LIN {X 0,Y 368.953,Z 167.528,A -85,B 0,C 180,E1 -12752.796,E2 -12752.796} C_VEL
LIN {X 0,Y 368.922,Z 167.518,A -85,B 0,C 180,E1 -12756.117,E2 -12756.117} C_VEL
LIN {X 0,Y 368.919,Z 167.528,A -85,B 0,C 180,E1 -12759.946,E2 -12759.946} C_VEL
LIN {X 0,Y 368.957,Z 167.521,A -85,B 0,C 180,E1 -12763.398,E2 -12763.398} C_VEL
LIN {X 0,Y 369.049,Z 167.51,A -85,B 0,C 180,E1 -12766.79,E2 -12766.79} C_VEL
LIN {X 0,Y 369.059,Z 167.505,A -85,B 0,C 180,E1 -12770.132,E2 -12770.132} C_VEL
LIN {X 0,Y 369.151,Z 167.503,A -85,B 0,C 180,E1 -12772.342,E2 -12772.342} C_VEL
LIN {X 0,Y 369.129,Z 167.493,A -85,B 0,C 180,E1 -12774.537,E2 -12774.537} C_VEL
LIN {X 0,Y 369.304,Z 167.479,A -85,B 0,C 180,E1 -12777.819,E2 -12777.819} C_VEL
LIN {X 0,Y 369.446,Z 167.464,A -85,B 0,C 180,E1 -12780,E2 -12780} C_VEL
LIN {X 0,Y 369.303,Z 167.47,A -85,B 0,C 180,E1 -12782.181,E2 -12782.181} C_VEL
LIN {X 0,Y 369.185,Z 167.495,A -85,B 0,C 180,E1 -12786.687,E2 -12786.687} C_VEL
LIN {X 0,Y 369.126,Z 167.489,A -85,B 0,C 180,E1 -12788.761,E2 -12788.761} C_VEL
LIN {X 0,Y 368.994,Z 167.52,A -85,B 0,C 180,E1 -12792.094,E2 -12792.094} C_VEL
LIN {X 0,Y 368.987,Z 167.509,A -85,B 0,C 180,E1 -12795.465,E2 -12795.465} C_VEL
LIN {X 0,Y 368.956,Z 167.525,A -85,B 0,C 180,E1 -12798.894,E2 -12798.894} C_VEL
LIN {X 0,Y 368.922,Z 167.521,A -85,B 0,C 180,E1 -12802.396,E2 -12802.396} C_VEL
LIN {X 0,Y 368.991,Z 167.523,A -85,B 0,C 180,E1 -12805.981,E2 -12805.981} C_VEL
LIN {X 0,Y 368.95,Z 167.523,A -85,B 0,C 180,E1 -12808.812,E2 -12808.812} C_VEL
LIN {X 0,Y 368.89,Z 167.526,A -85,B 0,C 180,E1 -12812.239,E2 -12812.239} C_VEL
LIN {X 0,Y 368.921,Z 167.494,A -85,B 0,C 180,E1 -12815.002,E2 -12815.002} C_VEL
LIN {X 0,Y 368.901,Z 167.532,A -85,B 0,C 180,E1 -12818.641,E2 -12818.641} C_VEL
LIN {X 0,Y 368.875,Z 167.52,A -85,B 0,C 180,E1 -12822.01,E2 -12822.01} C_VEL
LIN {X 0,Y 368.874,Z 167.527,A -85,B 0,C 180,E1 -12825.177,E2 -12825.177} C_VEL
LIN {X 0,Y 368.878,Z 167.529,A -85,B 0,C 180,E1 -12828.179,E2 -12828.179} C_VEL
LIN {X 0,Y 368.902,Z 167.522,A -85,B 0,C 180,E1 -12831.361,E2 -12831.361} C_VEL
LIN {X 0,Y 368.933,Z 167.516,A -85,B 0,C 180,E1 -12835.148,E2 -12835.148} C_VEL
LIN {X 0,Y 368.927,Z 167.52,A -85,B 0,C 180,E1 -12839.048,E2 -12839.048} C_VEL
LIN {X 0,Y 368.975,Z 167.527,A -85,B 0,C 180,E1 -12842.799,E2 -12842.799} C_VEL
LIN {X 0,Y 369.055,Z 167.91,A -85,B 0,C 180,E1 -12843.213,E2 -12843.213} C_VEL
LIN {X 0,Y 371.306,Z 179.09,A -85,B 0,C 180,E1 -12846.304,E2 -12846.304} C_VEL
LIN {X 0,Y 372.031,Z 183.742,A -85,B 0,C 180,E1 -12847.54,E2 -12847.54} C_VEL
LIN {X 0,Y 371.856,Z 187.412,A -85,B 0,C 180,E1 -12848.395,E2 -12848.395} C_VEL
LIN {X 0,Y 374.592,Z 201.248,A -85,B 0,C 180,E1 -12848.88,E2 -12848.88} C_VEL
LIN {X 0,Y 377.012,Z 215.027,A -85,B 0,C 180,E1 -12849.298,E2 -12849.298} C_VEL
LIN {X 0,Y 375.8,Z 295.344,A -85,B 0,C 180,E1 -12850.862,E2 -12850.862} C_VEL
LIN {X 0,Y 375.266,Z 308.388,A -85,B 0,C 180,E1 -12851.33,E2 -12851.33} C_VEL
LIN {X 0,Y 374.412,Z 321.526,A -85,B 0,C 180,E1 -12852.029,E2 -12852.029} C_VEL
LIN {X 0,Y 373.468,Z 333.374,A -85,B 0,C 180,E1 -12852.901,E2 -12852.901} C_VEL
LIN {X 0,Y 372.421,Z 345.135,A -85,B 0,C 180,E1 -12854.022,E2 -12854.022} C_VEL
LIN {X 0,Y 371.58,Z 354.998,A -85,B 0,C 180,E1 -12855.207,E2 -12855.207} C_VEL
LIN {X 0,Y 370.573,Z 364.199,A -85,B 0,C 180,E1 -12856.567,E2 -12856.567} C_VEL
LIN {X 0,Y 369.519,Z 373.137,A -85,B 0,C 180,E1 -12858.203,E2 -12858.203} C_VEL
LIN {X 0,Y 368.777,Z 380.334,A -85,B 0,C 180,E1 -12859.847,E2 -12859.847} C_VEL
LIN {X 0,Y 368.263,Z 385.189,A -85,B 0,C 180,E1 -12861.219,E2 -12861.219} C_VEL
LIN {X 0,Y 367.893,Z 389.907,A -85,B 0,C 180,E1 -12862.868,E2 -12862.868} C_VEL
LIN {X 0,Y 367.658,Z 393.52,A -85,B 0,C 180,E1 -12864.516,E2 -12864.516} C_VEL
LIN {X 0,Y 367.551,Z 395.387,A -85,B 0,C 180,E1 -12865.614,E2 -12865.614} C_VEL
LIN {X 0,Y 367.409,Z 396.793,A -85,B 0,C 180,E1 -12866.711,E2 -12866.711} C_VEL
LIN {X 0,Y 367.36,Z 398.408,A -85,B 0,C 180,E1 -12868.904,E2 -12868.904} C_VEL
LIN {X 0,Y 367.375,Z 398.642,A -85,B 0,C 180,E1 -12870,E2 -12870} C_VEL
LIN {X 0,Y 367.36,Z 398.452,A -85,B 0,C 180,E1 -12871.097,E2 -12871.097} C_VEL
LIN {X 0,Y 367.408,Z 396.893,A -85,B 0,C 180,E1 -12873.29,E2 -12873.29} C_VEL
LIN {X 0,Y 367.547,Z 395.53,A -85,B 0,C 180,E1 -12874.387,E2 -12874.387} C_VEL
LIN {X 0,Y 367.757,Z 391.844,A -85,B 0,C 180,E1 -12876.411,E2 -12876.411} C_VEL
LIN {X 0,Y 368.118,Z 387.186,A -85,B 0,C 180,E1 -12878.233,E2 -12878.233} C_VEL
LIN {X 0,Y 368.737,Z 380.727,A -85,B 0,C 180,E1 -12880.155,E2 -12880.155} C_VEL
LIN {X 0,Y 369.473,Z 373.632,A -85,B 0,C 180,E1 -12881.799,E2 -12881.799} C_VEL
LIN {X 0,Y 370.503,Z 364.792,A -85,B 0,C 180,E1 -12883.437,E2 -12883.437} C_VEL
LIN {X 0,Y 371.506,Z 356.065,A -85,B 0,C 180,E1 -12884.747,E2 -12884.747} C_VEL
LIN {X 0,Y 372.173,Z 347.371,A -85,B 0,C 180,E1 -12885.835,E2 -12885.835} C_VEL
LIN {X 0,Y 373.258,Z 336.1,A -85,B 0,C 180,E1 -12886.969,E2 -12886.969} C_VEL
LIN {X 0,Y 373.899,Z 328.987,A -85,B 0,C 180,E1 -12887.548,E2 -12887.548} C_VEL
LIN {X 0,Y 373.639,Z 323.72,A -85,B 0,C 180,E1 -12887.96,E2 -12887.96} C_VEL
LIN {X 0,Y 371.467,Z 315.053,A -85,B 0,C 180,E1 -12888.627,E2 -12888.627} C_VEL
LIN {X 0,Y 369.299,Z 306.135,A -85,B 0,C 180,E1 -12889.198,E2 -12889.198} C_VEL
LIN {X 0,Y 368.949,Z 300.482,A -85,B 0,C 180,E1 -12889.447,E2 -12889.447} C_VEL
LIN {X 0,Y 369.32,Z 287.934,A -85,B 0,C 180,E1 -12889.778,E2 -12889.778} C_VEL
LIN {X 0,Y 370.382,Z 215.345,A -85,B 0,C 180,E1 -12891.19,E2 -12891.19} C_VEL
LIN {X 0,Y 365.229,Z 188.64,A -85,B 0,C 180,E1 -12892.066,E2 -12892.066} C_VEL
LIN {X 0,Y 365.048,Z 187.088,A -85,B 0,C 180,E1 -12892.199,E2 -12892.199} C_VEL
LIN {X 0,Y 364.993,Z 184.101,A -85,B 0,C 180,E1 -12892.949,E2 -12892.949} C_VEL
LIN {X 0,Y 362.795,Z 172.573,A -85,B 0,C 180,E1 -12896.149,E2 -12896.149} C_VEL
LIN {X 0,Y 361.954,Z 168.46,A -85,B 0,C 180,E1 -12897.396,E2 -12897.396} C_VEL
LIN {X 0,Y 361.847,Z 168.401,A -85,B 0,C 180,E1 -12901.285,E2 -12901.285} C_VEL
LIN {X 0,Y 361.855,Z 168.4,A -85,B 0,C 180,E1 -12904.28,E2 -12904.28} C_VEL
LIN {X 0,Y 361.863,Z 168.409,A -85,B 0,C 180,E1 -12907.222,E2 -12907.222} C_VEL
LIN {X 0,Y 361.834,Z 168.395,A -85,B 0,C 180,E1 -12910.755,E2 -12910.755} C_VEL
LIN {X 0,Y 361.815,Z 168.411,A -85,B 0,C 180,E1 -12914.368,E2 -12914.368} C_VEL
LIN {X 0,Y 361.834,Z 168.391,A -85,B 0,C 180,E1 -12917.568,E2 -12917.568} C_VEL
LIN {X 0,Y 361.868,Z 168.407,A -85,B 0,C 180,E1 -12920.973,E2 -12920.973} C_VEL
LIN {X 0,Y 361.872,Z 168.37,A -85,B 0,C 180,E1 -12924.655,E2 -12924.655} C_VEL
LIN {X 0,Y 361.835,Z 168.412,A -85,B 0,C 180,E1 -12928.37,E2 -12928.37} C_VEL
LIN {X 0,Y 361.897,Z 168.401,A -85,B 0,C 180,E1 -12930.955,E2 -12930.955} C_VEL
LIN {X 0,Y 361.95,Z 168.391,A -85,B 0,C 180,E1 -12933.475,E2 -12933.475} C_VEL
LIN {X 0,Y 361.875,Z 168.402,A -85,B 0,C 180,E1 -12937.144,E2 -12937.144} C_VEL
LIN {X 0,Y 361.905,Z 168.402,A -85,B 0,C 180,E1 -12940.723,E2 -12940.723} C_VEL
LIN {X 0,Y 361.928,Z 168.396,A -85,B 0,C 180,E1 -12943.066,E2 -12943.066} C_VEL
LIN {X 0,Y 361.994,Z 168.389,A -85,B 0,C 180,E1 -12946.528,E2 -12946.528} C_VEL
LIN {X 0,Y 362.026,Z 168.376,A -85,B 0,C 180,E1 -12949.938,E2 -12949.938} C_VEL
LIN {X 0,Y 362.145,Z 168.369,A -85,B 0,C 180,E1 -12952.192,E2 -12952.192} C_VEL
LIN {X 0,Y 362.109,Z 168.376,A -85,B 0,C 180,E1 -12954.431,E2 -12954.431} C_VEL
LIN {X 0,Y 362.273,Z 168.345,A -85,B 0,C 180,E1 -12957.776,E2 -12957.776} C_VEL
LIN {X 0,Y 362.42,Z 168.339,A -85,B 0,C 180,E1 -12960,E2 -12960} C_VEL
LIN {X 0,Y 362.274,Z 168.354,A -85,B 0,C 180,E1 -12962.224,E2 -12962.224} C_VEL
LIN {X 0,Y 362.142,Z 168.369,A -85,B 0,C 180,E1 -12966.687,E2 -12966.687} C_VEL
LIN {X 0,Y 361.994,Z 168.384,A -85,B 0,C 180,E1 -12970.063,E2 -12970.063} C_VEL
LIN {X 0,Y 361.993,Z 168.392,A -85,B 0,C 180,E1 -12973.899,E2 -12973.899} C_VEL
LIN {X 0,Y 361.923,Z 168.395,A -85,B 0,C 180,E1 -12976.934,E2 -12976.934} C_VEL
LIN {X 0,Y 361.878,Z 168.405,A -85,B 0,C 180,E1 -12980.461,E2 -12980.461} C_VEL
LIN {X 0,Y 361.889,Z 168.395,A -85,B 0,C 180,E1 -12984.113,E2 -12984.113} C_VEL
LIN {X 0,Y 361.937,Z 168.4,A -85,B 0,C 180,E1 -12986.722,E2 -12986.722} C_VEL
LIN {X 0,Y 361.869,Z 168.402,A -85,B 0,C 180,E1 -12990.328,E2 -12990.328} C_VEL
LIN {X 0,Y 361.851,Z 168.402,A -85,B 0,C 180,E1 -12994.281,E2 -12994.281} C_VEL
LIN {X 0,Y 361.859,Z 168.38,A -85,B 0,C 180,E1 -12997.223,E2 -12997.223} C_VEL
LIN {X 0,Y 361.832,Z 168.415,A -85,B 0,C 180,E1 -13000.756,E2 -13000.756} C_VEL
LIN {X 0,Y 361.814,Z 168.412,A -85,B 0,C 180,E1 -13004.369,E2 -13004.369} C_VEL
LIN {X 0,Y 361.829,Z 168.412,A -85,B 0,C 180,E1 -13007.57,E2 -13007.57} C_VEL
LIN {X 0,Y 361.826,Z 168.396,A -85,B 0,C 180,E1 -13010.982,E2 -13010.982} C_VEL
LIN {X 0,Y 361.874,Z 168.408,A -85,B 0,C 180,E1 -13014.656,E2 -13014.656} C_VEL
LIN {X 0,Y 361.838,Z 168.412,A -85,B 0,C 180,E1 -13018.371,E2 -13018.371} C_VEL
LIN {X 0,Y 361.881,Z 168.545,A -85,B 0,C 180,E1 -13021.271,E2 -13021.271} C_VEL
LIN {X 0,Y 364.14,Z 179.165,A -85,B 0,C 180,E1 -13024.262,E2 -13024.262} C_VEL
LIN {X 0,Y 365.433,Z 186.328,A -85,B 0,C 180,E1 -13026.18,E2 -13026.18} C_VEL
LIN {X 0,Y 364.841,Z 193.578,A -85,B 0,C 180,E1 -13027.899,E2 -13027.899} C_VEL
LIN {X 0,Y 368.892,Z 215.373,A -85,B 0,C 180,E1 -13028.637,E2 -13028.637} C_VEL
LIN {X 0,Y 370.384,Z 225.055,A -85,B 0,C 180,E1 -13028.924,E2 -13028.924} C_VEL
LIN {X 0,Y 369.098,Z 301.362,A -85,B 0,C 180,E1 -13030.427,E2 -13030.427} C_VEL
LIN {X 0,Y 368.43,Z 314.558,A -85,B 0,C 180,E1 -13030.897,E2 -13030.897} C_VEL
LIN {X 0,Y 367.598,Z 326.674,A -85,B 0,C 180,E1 -13031.539,E2 -13031.539} C_VEL
LIN {X 0,Y 366.61,Z 338.9,A -85,B 0,C 180,E1 -13032.426,E2 -13032.426} C_VEL
LIN {X 0,Y 365.481,Z 350.464,A -85,B 0,C 180,E1 -13033.523,E2 -13033.523} C_VEL
LIN {X 0,Y 364.402,Z 361.281,A -85,B 0,C 180,E1 -13034.819,E2 -13034.819} C_VEL
LIN {X 0,Y 363.383,Z 371.057,A -85,B 0,C 180,E1 -13036.295,E2 -13036.295} C_VEL
LIN {X 0,Y 362.293,Z 379.964,A -85,B 0,C 180,E1 -13037.963,E2 -13037.963} C_VEL
LIN {X 0,Y 361.542,Z 387.13,A -85,B 0,C 180,E1 -13039.641,E2 -13039.641} C_VEL
LIN {X 0,Y 360.902,Z 393.654,A -85,B 0,C 180,E1 -13041.602,E2 -13041.602} C_VEL
LIN {X 0,Y 360.576,Z 397.97,A -85,B 0,C 180,E1 -13043.284,E2 -13043.284} C_VEL
LIN {X 0,Y 360.446,Z 400.254,A -85,B 0,C 180,E1 -13044.405,E2 -13044.405} C_VEL
LIN {X 0,Y 360.388,Z 402.105,A -85,B 0,C 180,E1 -13045.526,E2 -13045.526} C_VEL
LIN {X 0,Y 360.286,Z 403.492,A -85,B 0,C 180,E1 -13046.645,E2 -13046.645} C_VEL
LIN {X 0,Y 360.249,Z 405.086,A -85,B 0,C 180,E1 -13048.882,E2 -13048.882} C_VEL
LIN {X 0,Y 360.274,Z 405.299,A -85,B 0,C 180,E1 -13050,E2 -13050} C_VEL
LIN {X 0,Y 360.249,Z 405.081,A -85,B 0,C 180,E1 -13051.117,E2 -13051.117} C_VEL
LIN {X 0,Y 360.286,Z 403.483,A -85,B 0,C 180,E1 -13053.354,E2 -13053.354} C_VEL
LIN {X 0,Y 360.388,Z 402.092,A -85,B 0,C 180,E1 -13054.473,E2 -13054.473} C_VEL
LIN {X 0,Y 360.51,Z 399.158,A -85,B 0,C 180,E1 -13056.159,E2 -13056.159} C_VEL
LIN {X 0,Y 360.775,Z 395.206,A -85,B 0,C 180,E1 -13057.837,E2 -13057.837} C_VEL
LIN {X 0,Y 361.306,Z 389.114,A -85,B 0,C 180,E1 -13059.799,E2 -13059.799} C_VEL
LIN {X 0,Y 362.024,Z 382.458,A -85,B 0,C 180,E1 -13061.477,E2 -13061.477} C_VEL
LIN {X 0,Y 362.976,Z 374.197,A -85,B 0,C 180,E1 -13063.149,E2 -13063.149} C_VEL
LIN {X 0,Y 363.939,Z 365.725,A -85,B 0,C 180,E1 -13064.538,E2 -13064.538} C_VEL
LIN {X 0,Y 364.962,Z 355.253,A -85,B 0,C 180,E1 -13065.926,E2 -13065.926} C_VEL
LIN {X 0,Y 366.116,Z 343.462,A -85,B 0,C 180,E1 -13067.165,E2 -13067.165} C_VEL
LIN {X 0,Y 367.216,Z 331.594,A -85,B 0,C 180,E1 -13068.119,E2 -13068.119} C_VEL
LIN {X 0,Y 368.176,Z 319.239,A -85,B 0,C 180,E1 -13068.863,E2 -13068.863} C_VEL
LIN {X 0,Y 368.825,Z 306.535,A -85,B 0,C 180,E1 -13069.406,E2 -13069.406} C_VEL
LIN {X 0,Y 369.28,Z 293.176,A -85,B 0,C 180,E1 -13069.743,E2 -13069.743} C_VEL
LIN {X 0,Y 370.205,Z 223.387,A -85,B 0,C 180,E1 -13071.106,E2 -13071.106} C_VEL
LIN {X 0,Y 365.253,Z 196.039,A -85,B 0,C 180,E1 -13071.971,E2 -13071.971} C_VEL
LIN {X 0,Y 364.814,Z 193.463,A -85,B 0,C 180,E1 -13072.102,E2 -13072.102} C_VEL
LIN {X 0,Y 365.418,Z 186.266,A -85,B 0,C 180,E1 -13073.82,E2 -13073.82} C_VEL
LIN {X 0,Y 363.121,Z 174.181,A -85,B 0,C 180,E1 -13077.088,E2 -13077.088} C_VEL
LIN {X 0,Y 361.886,Z 168.471,A -85,B 0,C 180,E1 -13078.756,E2 -13078.756} C_VEL
LIN {X 0,Y 361.835,Z 168.413,A -85,B 0,C 180,E1 -13081.628,E2 -13081.628} C_VEL
LIN {X 0,Y 361.87,Z 168.409,A -85,B 0,C 180,E1 -13085.344,E2 -13085.344} C_VEL
LIN {X 0,Y 361.824,Z 168.397,A -85,B 0,C 180,E1 -13089.017,E2 -13089.017} C_VEL
LIN {X 0,Y 361.83,Z 168.409,A -85,B 0,C 180,E1 -13092.828,E2 -13092.828} C_VEL
LIN {X 0,Y 361.812,Z 168.411,A -85,B 0,C 180,E1 -13095.946,E2 -13095.946} C_VEL
LIN {X 0,Y 361.828,Z 168.415,A -85,B 0,C 180,E1 -13099.244,E2 -13099.244} C_VEL
LIN {X 0,Y 361.855,Z 168.38,A -85,B 0,C 180,E1 -13102.776,E2 -13102.776} C_VEL
LIN {X 0,Y 361.846,Z 168.404,A -85,B 0,C 180,E1 -13105.719,E2 -13105.719} C_VEL
LIN {X 0,Y 361.864,Z 168.402,A -85,B 0,C 180,E1 -13109.671,E2 -13109.671} C_VEL
LIN {X 0,Y 361.944,Z 168.398,A -85,B 0,C 180,E1 -13113.474,E2 -13113.474} C_VEL
LIN {X 0,Y 361.869,Z 168.405,A -85,B 0,C 180,E1 -13117.143,E2 -13117.143} C_VEL
LIN {X 0,Y 361.891,Z 168.4,A -85,B 0,C 180,E1 -13120.722,E2 -13120.722} C_VEL
LIN {X 0,Y 361.933,Z 168.397,A -85,B 0,C 180,E1 -13124.226,E2 -13124.226} C_VEL
LIN {X 0,Y 361.99,Z 168.392,A -85,B 0,C 180,E1 -13126.527,E2 -13126.527} C_VEL
LIN {X 0,Y 362.023,Z 168.381,A -85,B 0,C 180,E1 -13129.938,E2 -13129.938} C_VEL
LIN {X 0,Y 362.149,Z 168.368,A -85,B 0,C 180,E1 -13133.313,E2 -13133.313} C_VEL
LIN {X 0,Y 362.268,Z 168.355,A -85,B 0,C 180,E1 -13137.776,E2 -13137.776} C_VEL
LIN {X 0,Y 362.416,Z 168.34,A -85,B 0,C 180,E1 -13140,E2 -13140} C_VEL
LIN {X 0,Y 362.268,Z 168.346,A -85,B 0,C 180,E1 -13142.224,E2 -13142.224} C_VEL
LIN {X 0,Y 362.158,Z 168.37,A -85,B 0,C 180,E1 -13146.686,E2 -13146.686} C_VEL
LIN {X 0,Y 362.063,Z 168.368,A -85,B 0,C 180,E1 -13148.934,E2 -13148.934} C_VEL
LIN {X 0,Y 361.949,Z 168.4,A -85,B 0,C 180,E1 -13152.333,E2 -13152.333} C_VEL
LIN {X 0,Y 361.951,Z 168.388,A -85,B 0,C 180,E1 -13154.621,E2 -13154.621} C_VEL
LIN {X 0,Y 361.947,Z 168.397,A -85,B 0,C 180,E1 -13158.1,E2 -13158.1} C_VEL
LIN {X 0,Y 361.882,Z 168.398,A -85,B 0,C 180,E1 -13161.654,E2 -13161.654} C_VEL
LIN {X 0,Y 361.919,Z 168.401,A -85,B 0,C 180,E1 -13165.291,E2 -13165.291} C_VEL
LIN {X 0,Y 361.905,Z 168.395,A -85,B 0,C 180,E1 -13167.779,E2 -13167.779} C_VEL
LIN {X 0,Y 361.839,Z 168.41,A -85,B 0,C 180,E1 -13171.286,E2 -13171.286} C_VEL
LIN {X 0,Y 361.846,Z 168.379,A -85,B 0,C 180,E1 -13174.281,E2 -13174.281} C_VEL
LIN {X 0,Y 361.856,Z 168.396,A -85,B 0,C 180,E1 -13177.224,E2 -13177.224} C_VEL
LIN {X 0,Y 361.829,Z 168.409,A -85,B 0,C 180,E1 -13180.756,E2 -13180.756} C_VEL
LIN {X 0,Y 361.81,Z 168.396,A -85,B 0,C 180,E1 -13184.37,E2 -13184.37} C_VEL
LIN {X 0,Y 361.831,Z 168.415,A -85,B 0,C 180,E1 -13187.569,E2 -13187.569} C_VEL
LIN {X 0,Y 361.864,Z 168.394,A -85,B 0,C 180,E1 -13190.975,E2 -13190.975} C_VEL
LIN {X 0,Y 361.871,Z 168.397,A -85,B 0,C 180,E1 -13194.656,E2 -13194.656} C_VEL
LIN {X 0,Y 361.835,Z 168.405,A -85,B 0,C 180,E1 -13198.372,E2 -13198.372} C_VEL
LIN {X 0,Y 361.913,Z 168.401,A -85,B 0,C 180,E1 -13202.223,E2 -13202.223} C_VEL
LIN {X 0,Y 361.98,Z 168.589,A -85,B 0,C 180,E1 -13202.791,E2 -13202.791} C_VEL
LIN {X 0,Y 364.016,Z 178.714,A -85,B 0,C 180,E1 -13205.683,E2 -13205.683} C_VEL
LIN {X 0,Y 365.086,Z 185.481,A -85,B 0,C 180,E1 -13207.521,E2 -13207.521} C_VEL
LIN {X 0,Y 365.036,Z 187.672,A -85,B 0,C 180,E1 -13207.989,E2 -13207.989} C_VEL
LIN {X 0,Y 370.137,Z 213.867,A -85,B 0,C 180,E1 -13208.87,E2 -13208.87} C_VEL
LIN {X 0,Y 370.357,Z 219.609,A -85,B 0,C 180,E1 -13209,E2 -13209} C_VEL
LIN {X 0,Y 369.118,Z 295.425,A -85,B 0,C 180,E1 -13210.502,E2 -13210.502} C_VEL
LIN {X 0,Y 368.552,Z 308.464,A -85,B 0,C 180,E1 -13210.977,E2 -13210.977} C_VEL
LIN {X 0,Y 367.782,Z 320.497,A -85,B 0,C 180,E1 -13211.622,E2 -13211.622} C_VEL
LIN {X 0,Y 366.817,Z 331.857,A -85,B 0,C 180,E1 -13212.438,E2 -13212.438} C_VEL
LIN {X 0,Y 365.721,Z 343.786,A -85,B 0,C 180,E1 -13213.564,E2 -13213.564} C_VEL
LIN {X 0,Y 364.784,Z 354.024,A -85,B 0,C 180,E1 -13214.785,E2 -13214.785} C_VEL
LIN {X 0,Y 363.837,Z 362.569,A -85,B 0,C 180,E1 -13216.028,E2 -13216.028} C_VEL
LIN {X 0,Y 362.915,Z 370.46,A -85,B 0,C 180,E1 -13217.417,E2 -13217.417} C_VEL
LIN {X 0,Y 362.007,Z 378.174,A -85,B 0,C 180,E1 -13219.09,E2 -13219.09} C_VEL
LIN {X 0,Y 361.242,Z 385.256,A -85,B 0,C 180,E1 -13221.047,E2 -13221.047} C_VEL
LIN {X 0,Y 360.842,Z 389.973,A -85,B 0,C 180,E1 -13222.728,E2 -13222.728} C_VEL
LIN {X 0,Y 360.573,Z 393.586,A -85,B 0,C 180,E1 -13224.408,E2 -13224.408} C_VEL
LIN {X 0,Y 360.486,Z 395.452,A -85,B 0,C 180,E1 -13225.528,E2 -13225.528} C_VEL
LIN {X 0,Y 360.332,Z 396.859,A -85,B 0,C 180,E1 -13226.646,E2 -13226.646} C_VEL
LIN {X 0,Y 360.26,Z 398.474,A -85,B 0,C 180,E1 -13228.883,E2 -13228.883} C_VEL
LIN {X 0,Y 360.275,Z 398.707,A -85,B 0,C 180,E1 -13230,E2 -13230} C_VEL
LIN {X 0,Y 360.26,Z 398.517,A -85,B 0,C 180,E1 -13231.118,E2 -13231.118} C_VEL
LIN {X 0,Y 360.33,Z 396.958,A -85,B 0,C 180,E1 -13233.355,E2 -13233.355} C_VEL
LIN {X 0,Y 360.459,Z 395.595,A -85,B 0,C 180,E1 -13234.473,E2 -13234.473} C_VEL
LIN {X 0,Y 360.684,Z 392.187,A -85,B 0,C 180,E1 -13236.41,E2 -13236.41} C_VEL
LIN {X 0,Y 361.078,Z 387.25,A -85,B 0,C 180,E1 -13238.394,E2 -13238.394} C_VEL
LIN {X 0,Y 361.739,Z 380.79,A -85,B 0,C 180,E1 -13240.353,E2 -13240.353} C_VEL
LIN {X 0,Y 362.487,Z 373.695,A -85,B 0,C 180,E1 -13242.03,E2 -13242.03} C_VEL
LIN {X 0,Y 363.584,Z 364.854,A -85,B 0,C 180,E1 -13243.697,E2 -13243.697} C_VEL
LIN {X 0,Y 364.718,Z 355.058,A -85,B 0,C 180,E1 -13245.183,E2 -13245.183} C_VEL
LIN {X 0,Y 365.509,Z 345.747,A -85,B 0,C 180,E1 -13246.332,E2 -13246.332} C_VEL
LIN {X 0,Y 366.609,Z 334.579,A -85,B 0,C 180,E1 -13247.43,E2 -13247.43} C_VEL
LIN {X 0,Y 367.68,Z 322.048,A -85,B 0,C 180,E1 -13248.384,E2 -13248.384} C_VEL
LIN {X 0,Y 368.487,Z 309.138,A -85,B 0,C 180,E1 -13249.1,E2 -13249.1} C_VEL
LIN {X 0,Y 368.949,Z 300.482,A -85,B 0,C 180,E1 -13249.447,E2 -13249.447} C_VEL
LIN {X 0,Y 368.568,Z 294.756,A -85,B 0,C 180,E1 -13249.661,E2 -13249.661} C_VEL
LIN {X 0,Y 363.474,Z 276.11,A -85,B 0,C 180,E1 -13250.361,E2 -13250.361} C_VEL
LIN {X 0,Y 362.943,Z 270.294,A -85,B 0,C 180,E1 -13250.505,E2 -13250.505} C_VEL
LIN {X 0,Y 363.768,Z 216.155,A -85,B 0,C 180,E1 -13251.579,E2 -13251.579} C_VEL
LIN {X 0,Y 358.454,Z 188.842,A -85,B 0,C 180,E1 -13252.5,E2 -13252.5} C_VEL
LIN {X 0,Y 358.231,Z 187.146,A -85,B 0,C 180,E1 -13252.646,E2 -13252.646} C_VEL
LIN {X 0,Y 356.625,Z 177.642,A -85,B 0,C 180,E1 -13255.272,E2 -13255.272} C_VEL
LIN {X 0,Y 354.899,Z 169.377,A -85,B 0,C 180,E1 -13257.733,E2 -13257.733} C_VEL
LIN {X 0,Y 354.8,Z 169.28,A -85,B 0,C 180,E1 -13260.998,E2 -13260.998} C_VEL
LIN {X 0,Y 354.807,Z 169.285,A -85,B 0,C 180,E1 -13263.702,E2 -13263.702} C_VEL
LIN {X 0,Y 354.798,Z 169.287,A -85,B 0,C 180,E1 -13266.459,E2 -13266.459} C_VEL
LIN {X 0,Y 354.824,Z 169.267,A -85,B 0,C 180,E1 -13269.423,E2 -13269.423} C_VEL
LIN {X 0,Y 354.787,Z 169.29,A -85,B 0,C 180,E1 -13272.867,E2 -13272.867} C_VEL
LIN {X 0,Y 354.764,Z 169.27,A -85,B 0,C 180,E1 -13276.103,E2 -13276.103} C_VEL
LIN {X 0,Y 354.786,Z 169.286,A -85,B 0,C 180,E1 -13279.179,E2 -13279.179} C_VEL
LIN {X 0,Y 354.805,Z 169.278,A -85,B 0,C 180,E1 -13282.402,E2 -13282.402} C_VEL
LIN {X 0,Y 354.809,Z 169.248,A -85,B 0,C 180,E1 -13284.94,E2 -13284.94} C_VEL
LIN {X 0,Y 354.79,Z 169.29,A -85,B 0,C 180,E1 -13288.405,E2 -13288.405} C_VEL
LIN {X 0,Y 354.846,Z 169.278,A -85,B 0,C 180,E1 -13291.618,E2 -13291.618} C_VEL
LIN {X 0,Y 354.894,Z 169.279,A -85,B 0,C 180,E1 -13294.172,E2 -13294.172} C_VEL
LIN {X 0,Y 354.811,Z 169.277,A -85,B 0,C 180,E1 -13297.892,E2 -13297.892} C_VEL
LIN {X 0,Y 354.919,Z 169.273,A -85,B 0,C 180,E1 -13301.891,E2 -13301.891} C_VEL
LIN {X 0,Y 354.938,Z 169.269,A -85,B 0,C 180,E1 -13305.981,E2 -13305.981} C_VEL
LIN {X 0,Y 354.972,Z 169.256,A -85,B 0,C 180,E1 -13309.736,E2 -13309.736} C_VEL
LIN {X 0,Y 355.108,Z 169.243,A -85,B 0,C 180,E1 -13312.037,E2 -13312.037} C_VEL
LIN {X 0,Y 355.084,Z 169.251,A -85,B 0,C 180,E1 -13314.32,E2 -13314.32} C_VEL
LIN {X 0,Y 355.236,Z 169.221,A -85,B 0,C 180,E1 -13317.732,E2 -13317.732} C_VEL
LIN {X 0,Y 355.369,Z 169.218,A -85,B 0,C 180,E1 -13320,E2 -13320} C_VEL
LIN {X 0,Y 355.237,Z 169.231,A -85,B 0,C 180,E1 -13322.268,E2 -13322.268} C_VEL
LIN {X 0,Y 355.105,Z 169.246,A -85,B 0,C 180,E1 -13326.82,E2 -13326.82} C_VEL
LIN {X 0,Y 354.95,Z 169.261,A -85,B 0,C 180,E1 -13330.265,E2 -13330.265} C_VEL
LIN {X 0,Y 354.938,Z 169.271,A -85,B 0,C 180,E1 -13334.019,E2 -13334.019} C_VEL
LIN {X 0,Y 354.885,Z 169.266,A -85,B 0,C 180,E1 -13338.092,E2 -13338.092} C_VEL
LIN {X 0,Y 354.811,Z 169.284,A -85,B 0,C 180,E1 -13342.108,E2 -13342.108} C_VEL
LIN {X 0,Y 354.894,Z 169.277,A -85,B 0,C 180,E1 -13345.828,E2 -13345.828} C_VEL
LIN {X 0,Y 354.814,Z 169.28,A -85,B 0,C 180,E1 -13349.682,E2 -13349.682} C_VEL
LIN {X 0,Y 354.803,Z 169.281,A -85,B 0,C 180,E1 -13353.702,E2 -13353.702} C_VEL
LIN {X 0,Y 354.794,Z 169.256,A -85,B 0,C 180,E1 -13356.46,E2 -13356.46} C_VEL
LIN {X 0,Y 354.822,Z 169.283,A -85,B 0,C 180,E1 -13359.424,E2 -13359.424} C_VEL
LIN {X 0,Y 354.785,Z 169.284,A -85,B 0,C 180,E1 -13362.867,E2 -13362.867} C_VEL
LIN {X 0,Y 354.764,Z 169.292,A -85,B 0,C 180,E1 -13366.104,E2 -13366.104} C_VEL
LIN {X 0,Y 354.78,Z 169.291,A -85,B 0,C 180,E1 -13369.178,E2 -13369.178} C_VEL
LIN {X 0,Y 354.799,Z 169.274,A -85,B 0,C 180,E1 -13372.404,E2 -13372.404} C_VEL
LIN {X 0,Y 354.811,Z 169.283,A -85,B 0,C 180,E1 -13374.941,E2 -13374.941} C_VEL
LIN {X 0,Y 354.794,Z 169.289,A -85,B 0,C 180,E1 -13378.405,E2 -13378.405} C_VEL
LIN {X 0,Y 354.842,Z 169.383,A -85,B 0,C 180,E1 -13380.883,E2 -13380.883} C_VEL
LIN {X 0,Y 357.171,Z 180.29,A -85,B 0,C 180,E1 -13384.036,E2 -13384.036} C_VEL
LIN {X 0,Y 358.462,Z 187.453,A -85,B 0,C 180,E1 -13385.995,E2 -13385.995} C_VEL
LIN {X 0,Y 358.046,Z 193.292,A -85,B 0,C 180,E1 -13387.429,E2 -13387.429} C_VEL
LIN {X 0,Y 358.746,Z 197.435,A -85,B 0,C 180,E1 -13387.623,E2 -13387.623} C_VEL
LIN {X 0,Y 363.292,Z 222.248,A -85,B 0,C 180,E1 -13388.435,E2 -13388.435} C_VEL
LIN {X 0,Y 363.756,Z 226.414,A -85,B 0,C 180,E1 -13388.55,E2 -13388.55} C_VEL
LIN {X 0,Y 362.423,Z 301.31,A -85,B 0,C 180,E1 -13390.052,E2 -13390.052} C_VEL
LIN {X 0,Y 361.734,Z 314.502,A -85,B 0,C 180,E1 -13390.529,E2 -13390.529} C_VEL
LIN {X 0,Y 360.875,Z 326.615,A -85,B 0,C 180,E1 -13391.183,E2 -13391.183} C_VEL
LIN {X 0,Y 359.841,Z 338.839,A -85,B 0,C 180,E1 -13392.085,E2 -13392.085} C_VEL
LIN {X 0,Y 358.669,Z 350.403,A -85,B 0,C 180,E1 -13393.201,E2 -13393.201} C_VEL
LIN {X 0,Y 357.539,Z 361.219,A -85,B 0,C 180,E1 -13394.521,E2 -13394.521} C_VEL
LIN {X 0,Y 356.484,Z 370.994,A -85,B 0,C 180,E1 -13396.024,E2 -13396.024} C_VEL
LIN {X 0,Y 355.311,Z 379.9,A -85,B 0,C 180,E1 -13397.723,E2 -13397.723} C_VEL
LIN {X 0,Y 354.521,Z 387.066,A -85,B 0,C 180,E1 -13399.434,E2 -13399.434} C_VEL
LIN {X 0,Y 353.853,Z 393.59,A -85,B 0,C 180,E1 -13401.433,E2 -13401.433} C_VEL
LIN {X 0,Y 353.509,Z 397.905,A -85,B 0,C 180,E1 -13403.149,E2 -13403.149} C_VEL
LIN {X 0,Y 353.357,Z 400.19,A -85,B 0,C 180,E1 -13404.292,E2 -13404.292} C_VEL
LIN {X 0,Y 353.303,Z 402.041,A -85,B 0,C 180,E1 -13405.436,E2 -13405.436} C_VEL
LIN {X 0,Y 353.211,Z 403.428,A -85,B 0,C 180,E1 -13406.577,E2 -13406.577} C_VEL
LIN {X 0,Y 353.148,Z 405.021,A -85,B 0,C 180,E1 -13408.859,E2 -13408.859} C_VEL
LIN {X 0,Y 353.175,Z 405.234,A -85,B 0,C 180,E1 -13410,E2 -13410} C_VEL
LIN {X 0,Y 353.148,Z 405.016,A -85,B 0,C 180,E1 -13411.14,E2 -13411.14} C_VEL
LIN {X 0,Y 353.21,Z 403.418,A -85,B 0,C 180,E1 -13413.422,E2 -13413.422} C_VEL
LIN {X 0,Y 353.303,Z 402.026,A -85,B 0,C 180,E1 -13414.563,E2 -13414.563} C_VEL
LIN {X 0,Y 353.434,Z 399.342,A -85,B 0,C 180,E1 -13416.149,E2 -13416.149} C_VEL
LIN {X 0,Y 353.723,Z 395.14,A -85,B 0,C 180,E1 -13417.994,E2 -13417.994} C_VEL
LIN {X 0,Y 354.29,Z 389.048,A -85,B 0,C 180,E1 -13419.995,E2 -13419.995} C_VEL
LIN {X 0,Y 355.022,Z 382.391,A -85,B 0,C 180,E1 -13421.706,E2 -13421.706} C_VEL
LIN {X 0,Y 356.048,Z 374.13,A -85,B 0,C 180,E1 -13423.41,E2 -13423.41} C_VEL
LIN {X 0,Y 357.043,Z 365.658,A -85,B 0,C 180,E1 -13424.825,E2 -13424.825} C_VEL
LIN {X 0,Y 358.13,Z 355.185,A -85,B 0,C 180,E1 -13426.238,E2 -13426.238} C_VEL
LIN {X 0,Y 359.339,Z 343.393,A -85,B 0,C 180,E1 -13427.499,E2 -13427.499} C_VEL
LIN {X 0,Y 360.483,Z 331.523,A -85,B 0,C 180,E1 -13428.469,E2 -13428.469} C_VEL
LIN {X 0,Y 361.446,Z 319.166,A -85,B 0,C 180,E1 -13429.227,E2 -13429.227} C_VEL
LIN {X 0,Y 362.133,Z 306.459,A -85,B 0,C 180,E1 -13429.779,E2 -13429.779} C_VEL
LIN {X 0,Y 362.612,Z 293.091,A -85,B 0,C 180,E1 -13430.121,E2 -13430.121} C_VEL
LIN {X 0,Y 363.594,Z 224.394,A -85,B 0,C 180,E1 -13431.486,E2 -13431.486} C_VEL
LIN {X 0,Y 358.821,Z 197.843,A -85,B 0,C 180,E1 -13432.346,E2 -13432.346} C_VEL
LIN {X 0,Y 358.017,Z 193.627,A -85,B 0,C 180,E1 -13432.516,E2 -13432.516} C_VEL
LIN {X 0,Y 358.48,Z 188.58,A -85,B 0,C 180,E1 -13433.696,E2 -13433.696} C_VEL
LIN {X 0,Y 357.359,Z 181.416,A -85,B 0,C 180,E1 -13435.635,E2 -13435.635} C_VEL
LIN {X 0,Y 355.129,Z 170.735,A -85,B 0,C 180,E1 -13438.657,E2 -13438.657} C_VEL
LIN {X 0,Y 354.808,Z 169.313,A -85,B 0,C 180,E1 -13439.152,E2 -13439.152} C_VEL
LIN {X 0,Y 354.784,Z 169.294,A -85,B 0,C 180,E1 -13442.332,E2 -13442.332} C_VEL
LIN {X 0,Y 354.818,Z 169.289,A -85,B 0,C 180,E1 -13445.698,E2 -13445.698} C_VEL
LIN {X 0,Y 354.794,Z 169.276,A -85,B 0,C 180,E1 -13449.417,E2 -13449.417} C_VEL
LIN {X 0,Y 354.782,Z 169.287,A -85,B 0,C 180,E1 -13452.866,E2 -13452.866} C_VEL
LIN {X 0,Y 354.76,Z 169.289,A -85,B 0,C 180,E1 -13456.102,E2 -13456.102} C_VEL
LIN {X 0,Y 354.781,Z 169.293,A -85,B 0,C 180,E1 -13459.178,E2 -13459.178} C_VEL
LIN {X 0,Y 354.799,Z 169.261,A -85,B 0,C 180,E1 -13462.402,E2 -13462.402} C_VEL
LIN {X 0,Y 354.803,Z 169.266,A -85,B 0,C 180,E1 -13464.94,E2 -13464.94} C_VEL
LIN {X 0,Y 354.785,Z 169.291,A -85,B 0,C 180,E1 -13468.404,E2 -13468.404} C_VEL
LIN {X 0,Y 354.837,Z 169.281,A -85,B 0,C 180,E1 -13471.618,E2 -13471.618} C_VEL
LIN {X 0,Y 354.888,Z 169.277,A -85,B 0,C 180,E1 -13474.172,E2 -13474.172} C_VEL
LIN {X 0,Y 354.805,Z 169.285,A -85,B 0,C 180,E1 -13477.892,E2 -13477.892} C_VEL
LIN {X 0,Y 354.879,Z 169.266,A -85,B 0,C 180,E1 -13481.907,E2 -13481.907} C_VEL
LIN {X 0,Y 354.933,Z 169.271,A -85,B 0,C 180,E1 -13485.981,E2 -13485.981} C_VEL
LIN {X 0,Y 354.97,Z 169.259,A -85,B 0,C 180,E1 -13489.736,E2 -13489.736} C_VEL
LIN {X 0,Y 355.114,Z 169.245,A -85,B 0,C 180,E1 -13493.18,E2 -13493.18} C_VEL
LIN {X 0,Y 355.231,Z 169.232,A -85,B 0,C 180,E1 -13497.732,E2 -13497.732} C_VEL
LIN {X 0,Y 355.385,Z 169.215,A -85,B 0,C 180,E1 -13500,E2 -13500} C_VEL
LIN {X 0,Y 355.231,Z 169.222,A -85,B 0,C 180,E1 -13502.268,E2 -13502.268} C_VEL
LIN {X 0,Y 355.125,Z 169.245,A -85,B 0,C 180,E1 -13506.82,E2 -13506.82} C_VEL
LIN {X 0,Y 355.004,Z 169.246,A -85,B 0,C 180,E1 -13509.113,E2 -13509.113} C_VEL
LIN {X 0,Y 354.91,Z 169.276,A -85,B 0,C 180,E1 -13512.581,E2 -13512.581} C_VEL
LIN {X 0,Y 354.879,Z 169.266,A -85,B 0,C 180,E1 -13516.097,E2 -13516.097} C_VEL
LIN {X 0,Y 354.893,Z 169.28,A -85,B 0,C 180,E1 -13518.473,E2 -13518.473} C_VEL
LIN {X 0,Y 354.825,Z 169.276,A -85,B 0,C 180,E1 -13522.107,E2 -13522.107} C_VEL
LIN {X 0,Y 354.89,Z 169.279,A -85,B 0,C 180,E1 -13525.828,E2 -13525.828} C_VEL
LIN {X 0,Y 354.845,Z 169.281,A -85,B 0,C 180,E1 -13529.68,E2 -13529.68} C_VEL
LIN {X 0,Y 354.799,Z 169.264,A -85,B 0,C 180,E1 -13533.703,E2 -13533.703} C_VEL
LIN {X 0,Y 354.79,Z 169.262,A -85,B 0,C 180,E1 -13536.461,E2 -13536.461} C_VEL
LIN {X 0,Y 354.818,Z 169.286,A -85,B 0,C 180,E1 -13539.425,E2 -13539.425} C_VEL
LIN {X 0,Y 354.782,Z 169.267,A -85,B 0,C 180,E1 -13542.868,E2 -13542.868} C_VEL
LIN {X 0,Y 354.762,Z 169.293,A -85,B 0,C 180,E1 -13546.105,E2 -13546.105} C_VEL
LIN {X 0,Y 354.782,Z 169.276,A -85,B 0,C 180,E1 -13549.18,E2 -13549.18} C_VEL
LIN {X 0,Y 354.803,Z 169.29,A -85,B 0,C 180,E1 -13552.404,E2 -13552.404} C_VEL
LIN {X 0,Y 354.809,Z 169.275,A -85,B 0,C 180,E1 -13554.942,E2 -13554.942} C_VEL
LIN {X 0,Y 354.791,Z 169.282,A -85,B 0,C 180,E1 -13558.406,E2 -13558.406} C_VEL
LIN {X 0,Y 354.848,Z 169.278,A -85,B 0,C 180,E1 -13561.62,E2 -13561.62} C_VEL
LIN {X 0,Y 354.92,Z 169.503,A -85,B 0,C 180,E1 -13562.446,E2 -13562.446} C_VEL
LIN {X 0,Y 357.111,Z 180.301,A -85,B 0,C 180,E1 -13565.59,E2 -13565.59} C_VEL
LIN {X 0,Y 358.159,Z 187.07,A -85,B 0,C 180,E1 -13567.439,E2 -13567.439} C_VEL
LIN {X 0,Y 358.218,Z 187.932,A -85,B 0,C 180,E1 -13567.561,E2 -13567.561} C_VEL
LIN {X 0,Y 363.054,Z 212.192,A -85,B 0,C 180,E1 -13568.4,E2 -13568.4} C_VEL
LIN {X 0,Y 363.803,Z 217.381,A -85,B 0,C 180,E1 -13568.555,E2 -13568.555} C_VEL
LIN {X 0,Y 362.454,Z 295.506,A -85,B 0,C 180,E1 -13570.128,E2 -13570.128} C_VEL
LIN {X 0,Y 361.839,Z 308.539,A -85,B 0,C 180,E1 -13570.61,E2 -13570.61} C_VEL
LIN {X 0,Y 361.043,Z 320.57,A -85,B 0,C 180,E1 -13571.266,E2 -13571.266} C_VEL
LIN {X 0,Y 360.059,Z 331.928,A -85,B 0,C 180,E1 -13572.097,E2 -13572.097} C_VEL
LIN {X 0,Y 358.919,Z 343.855,A -85,B 0,C 180,E1 -13573.243,E2 -13573.243} C_VEL
LIN {X 0,Y 357.921,Z 353.931,A -85,B 0,C 180,E1 -13574.464,E2 -13574.464} C_VEL
LIN {X 0,Y 356.953,Z 362.637,A -85,B 0,C 180,E1 -13575.753,E2 -13575.753} C_VEL
LIN {X 0,Y 355.977,Z 370.527,A -85,B 0,C 180,E1 -13577.168,E2 -13577.168} C_VEL
LIN {X 0,Y 355.024,Z 378.241,A -85,B 0,C 180,E1 -13578.872,E2 -13578.872} C_VEL
LIN {X 0,Y 354.447,Z 383.507,A -85,B 0,C 180,E1 -13580.298,E2 -13580.298} C_VEL
LIN {X 0,Y 353.911,Z 388.617,A -85,B 0,C 180,E1 -13582.01,E2 -13582.01} C_VEL
LIN {X 0,Y 353.591,Z 392.373,A -85,B 0,C 180,E1 -13583.621,E2 -13583.621} C_VEL
LIN {X 0,Y 353.4,Z 395.518,A -85,B 0,C 180,E1 -13585.438,E2 -13585.438} C_VEL
LIN {X 0,Y 353.257,Z 396.924,A -85,B 0,C 180,E1 -13586.579,E2 -13586.579} C_VEL
LIN {X 0,Y 353.16,Z 398.539,A -85,B 0,C 180,E1 -13588.86,E2 -13588.86} C_VEL
LIN {X 0,Y 353.176,Z 398.772,A -85,B 0,C 180,E1 -13590,E2 -13590} C_VEL
LIN {X 0,Y 353.16,Z 398.582,A -85,B 0,C 180,E1 -13591.141,E2 -13591.141} C_VEL
LIN {X 0,Y 353.254,Z 397.022,A -85,B 0,C 180,E1 -13593.422,E2 -13593.422} C_VEL
LIN {X 0,Y 353.375,Z 395.659,A -85,B 0,C 180,E1 -13594.563,E2 -13594.563} C_VEL
LIN {X 0,Y 353.612,Z 392.524,A -85,B 0,C 180,E1 -13596.41,E2 -13596.41} C_VEL
LIN {X 0,Y 353.911,Z 388.877,A -85,B 0,C 180,E1 -13597.991,E2 -13597.991} C_VEL
LIN {X 0,Y 354.414,Z 383.842,A -85,B 0,C 180,E1 -13599.704,E2 -13599.704} C_VEL
LIN {X 0,Y 355.156,Z 377.506,A -85,B 0,C 180,E1 -13601.414,E2 -13601.414} C_VEL
LIN {X 0,Y 356.068,Z 369.577,A -85,B 0,C 180,E1 -13603.12,E2 -13603.12} C_VEL
LIN {X 0,Y 357.324,Z 359.715,A -85,B 0,C 180,E1 -13604.815,E2 -13604.815} C_VEL
LIN {X 0,Y 358.342,Z 349.369,A -85,B 0,C 180,E1 -13606.229,E2 -13606.229} C_VEL
LIN {X 0,Y 359.401,Z 339.122,A -85,B 0,C 180,E1 -13607.35,E2 -13607.35} C_VEL
LIN {X 0,Y 360.473,Z 327.912,A -85,B 0,C 180,E1 -13608.324,E2 -13608.324} C_VEL
LIN {X 0,Y 361.419,Z 315.287,A -85,B 0,C 180,E1 -13609.156,E2 -13609.156} C_VEL
LIN {X 0,Y 362.203,Z 301.718,A -85,B 0,C 180,E1 -13609.776,E2 -13609.776} C_VEL
LIN {X 0,Y 362.624,Z 289.635,A -85,B 0,C 180,E1 -13610.121,E2 -13610.121} C_VEL
LIN {X 0,Y 362.943,Z 270.294,A -85,B 0,C 180,E1 -13610.505,E2 -13610.505} C_VEL
LIN {X 0,Y 362.432,Z 264.482,A -85,B 0,C 180,E1 -13610.656,E2 -13610.656} C_VEL
LIN {X 0,Y 357.364,Z 245.796,A -85,B 0,C 180,E1 -13611.358,E2 -13611.358} C_VEL
LIN {X 0,Y 356.842,Z 239.985,A -85,B 0,C 180,E1 -13611.514,E2 -13611.514} C_VEL
LIN {X 0,Y 357.225,Z 217.327,A -85,B 0,C 180,E1 -13611.97,E2 -13611.97} C_VEL
LIN {X 0,Y 351.764,Z 189.499,A -85,B 0,C 180,E1 -13612.933,E2 -13612.933} C_VEL
LIN {X 0,Y 351.211,Z 187.405,A -85,B 0,C 180,E1 -13613.083,E2 -13613.083} C_VEL
LIN {X 0,Y 349.319,Z 177.174,A -85,B 0,C 180,E1 -13615.987,E2 -13615.987} C_VEL
LIN {X 0,Y 347.843,Z 170.212,A -85,B 0,C 180,E1 -13618.141,E2 -13618.141} C_VEL
LIN {X 0,Y 347.745,Z 170.159,A -85,B 0,C 180,E1 -13621.699,E2 -13621.699} C_VEL
LIN {X 0,Y 347.745,Z 170.155,A -85,B 0,C 180,E1 -13624.464,E2 -13624.464} C_VEL
LIN {X 0,Y 347.773,Z 170.162,A -85,B 0,C 180,E1 -13627.988,E2 -13627.988} C_VEL
LIN {X 0,Y 347.75,Z 170.159,A -85,B 0,C 180,E1 -13631.83,E2 -13631.83} C_VEL
LIN {X 0,Y 347.704,Z 170.164,A -85,B 0,C 180,E1 -13635.026,E2 -13635.026} C_VEL
LIN {X 0,Y 347.749,Z 170.154,A -85,B 0,C 180,E1 -13638.397,E2 -13638.397} C_VEL
LIN {X 0,Y 347.772,Z 170.158,A -85,B 0,C 180,E1 -13642.011,E2 -13642.011} C_VEL
LIN {X 0,Y 347.742,Z 170.129,A -85,B 0,C 180,E1 -13645.536,E2 -13645.536} C_VEL
LIN {X 0,Y 347.761,Z 170.167,A -85,B 0,C 180,E1 -13649.653,E2 -13649.653} C_VEL
LIN {X 0,Y 347.847,Z 170.146,A -85,B 0,C 180,E1 -13652.745,E2 -13652.745} C_VEL
LIN {X 0,Y 347.781,Z 170.16,A -85,B 0,C 180,E1 -13656.161,E2 -13656.161} C_VEL
LIN {X 0,Y 347.802,Z 170.159,A -85,B 0,C 180,E1 -13659.909,E2 -13659.909} C_VEL
LIN {X 0,Y 347.862,Z 170.148,A -85,B 0,C 180,E1 -13662.359,E2 -13662.359} C_VEL
LIN {X 0,Y 347.893,Z 170.145,A -85,B 0,C 180,E1 -13665.971,E2 -13665.971} C_VEL
LIN {X 0,Y 347.923,Z 170.137,A -85,B 0,C 180,E1 -13669.525,E2 -13669.525} C_VEL
LIN {X 0,Y 348.099,Z 170.118,A -85,B 0,C 180,E1 -13673.042,E2 -13673.042} C_VEL
LIN {X 0,Y 348.198,Z 170.097,A -85,B 0,C 180,E1 -13677.686,E2 -13677.686} C_VEL
LIN {X 0,Y 348.319,Z 170.096,A -85,B 0,C 180,E1 -13680,E2 -13680} C_VEL
LIN {X 0,Y 348.199,Z 170.107,A -85,B 0,C 180,E1 -13682.313,E2 -13682.313} C_VEL
LIN {X 0,Y 348.071,Z 170.123,A -85,B 0,C 180,E1 -13686.958,E2 -13686.958} C_VEL
LIN {X 0,Y 347.891,Z 170.14,A -85,B 0,C 180,E1 -13690.476,E2 -13690.476} C_VEL
LIN {X 0,Y 347.894,Z 170.148,A -85,B 0,C 180,E1 -13694.15,E2 -13694.15} C_VEL
LIN {X 0,Y 347.825,Z 170.145,A -85,B 0,C 180,E1 -13698.259,E2 -13698.259} C_VEL
LIN {X 0,Y 347.763,Z 170.164,A -85,B 0,C 180,E1 -13701.626,E2 -13701.626} C_VEL
LIN {X 0,Y 347.807,Z 170.154,A -85,B 0,C 180,E1 -13705.109,E2 -13705.109} C_VEL
LIN {X 0,Y 347.804,Z 170.157,A -85,B 0,C 180,E1 -13707.694,E2 -13707.694} C_VEL
LIN {X 0,Y 347.746,Z 170.161,A -85,B 0,C 180,E1 -13710.348,E2 -13710.348} C_VEL
LIN {X 0,Y 347.745,Z 170.159,A -85,B 0,C 180,E1 -13714.044,E2 -13714.044} C_VEL
LIN {X 0,Y 347.758,Z 170.135,A -85,B 0,C 180,E1 -13717.321,E2 -13717.321} C_VEL
LIN {X 0,Y 347.729,Z 170.168,A -85,B 0,C 180,E1 -13720.298,E2 -13720.298} C_VEL
LIN {X 0,Y 347.721,Z 170.164,A -85,B 0,C 180,E1 -13723.409,E2 -13723.409} C_VEL
LIN {X 0,Y 347.723,Z 170.166,A -85,B 0,C 180,E1 -13726.687,E2 -13726.687} C_VEL
LIN {X 0,Y 347.726,Z 170.162,A -85,B 0,C 180,E1 -13730.177,E2 -13730.177} C_VEL
LIN {X 0,Y 347.756,Z 170.154,A -85,B 0,C 180,E1 -13732.679,E2 -13732.679} C_VEL
LIN {X 0,Y 347.748,Z 170.155,A -85,B 0,C 180,E1 -13735.957,E2 -13735.957} C_VEL
LIN {X 0,Y 347.741,Z 170.161,A -85,B 0,C 180,E1 -13739.652,E2 -13739.652} C_VEL
LIN {X 0,Y 347.797,Z 170.349,A -85,B 0,C 180,E1 -13740.545,E2 -13740.545} C_VEL
LIN {X 0,Y 350.193,Z 181.415,A -85,B 0,C 180,E1 -13743.799,E2 -13743.799} C_VEL
LIN {X 0,Y 351.564,Z 189.769,A -85,B 0,C 180,E1 -13746.121,E2 -13746.121} C_VEL
LIN {X 0,Y 351.258,Z 193.32,A -85,B 0,C 180,E1 -13746.981,E2 -13746.981} C_VEL
LIN {X 0,Y 352.373,Z 199.522,A -85,B 0,C 180,E1 -13747.242,E2 -13747.242} C_VEL
LIN {X 0,Y 356.912,Z 224.52,A -85,B 0,C 180,E1 -13748.079,E2 -13748.079} C_VEL
LIN {X 0,Y 357.075,Z 229.998,A -85,B 0,C 180,E1 -13748.205,E2 -13748.205} C_VEL
LIN {X 0,Y 355.772,Z 301.258,A -85,B 0,C 180,E1 -13749.662,E2 -13749.662} C_VEL
LIN {X 0,Y 355.039,Z 314.445,A -85,B 0,C 180,E1 -13750.147,E2 -13750.147} C_VEL
LIN {X 0,Y 354.148,Z 326.557,A -85,B 0,C 180,E1 -13750.811,E2 -13750.811} C_VEL
LIN {X 0,Y 353.094,Z 338.779,A -85,B 0,C 180,E1 -13751.73,E2 -13751.73} C_VEL
LIN {X 0,Y 351.88,Z 350.342,A -85,B 0,C 180,E1 -13752.867,E2 -13752.867} C_VEL
LIN {X 0,Y 350.679,Z 361.24,A -85,B 0,C 180,E1 -13754.222,E2 -13754.222} C_VEL
LIN {X 0,Y 349.576,Z 370.931,A -85,B 0,C 180,E1 -13755.742,E2 -13755.742} C_VEL
LIN {X 0,Y 348.353,Z 379.837,A -85,B 0,C 180,E1 -13757.474,E2 -13757.474} C_VEL
LIN {X 0,Y 347.526,Z 387.002,A -85,B 0,C 180,E1 -13759.218,E2 -13759.218} C_VEL
LIN {X 0,Y 346.97,Z 391.838,A -85,B 0,C 180,E1 -13760.674,E2 -13760.674} C_VEL
LIN {X 0,Y 346.527,Z 396.537,A -85,B 0,C 180,E1 -13762.424,E2 -13762.424} C_VEL
LIN {X 0,Y 346.289,Z 400.126,A -85,B 0,C 180,E1 -13764.175,E2 -13764.175} C_VEL
LIN {X 0,Y 346.221,Z 401.976,A -85,B 0,C 180,E1 -13765.342,E2 -13765.342} C_VEL
LIN {X 0,Y 346.137,Z 403.363,A -85,B 0,C 180,E1 -13766.507,E2 -13766.507} C_VEL
LIN {X 0,Y 346.051,Z 404.956,A -85,B 0,C 180,E1 -13768.836,E2 -13768.836} C_VEL
LIN {X 0,Y 346.075,Z 405.169,A -85,B 0,C 180,E1 -13769.999,E2 -13769.999} C_VEL
LIN {X 0,Y 346.051,Z 404.951,A -85,B 0,C 180,E1 -13771.163,E2 -13771.163} C_VEL
LIN {X 0,Y 346.137,Z 403.353,A -85,B 0,C 180,E1 -13773.492,E2 -13773.492} C_VEL
LIN {X 0,Y 346.221,Z 401.961,A -85,B 0,C 180,E1 -13774.657,E2 -13774.657} C_VEL
LIN {X 0,Y 346.325,Z 399.623,A -85,B 0,C 180,E1 -13776.086,E2 -13776.086} C_VEL
LIN {X 0,Y 346.667,Z 395.074,A -85,B 0,C 180,E1 -13778.158,E2 -13778.158} C_VEL
LIN {X 0,Y 347.282,Z 388.981,A -85,B 0,C 180,E1 -13780.199,E2 -13780.199} C_VEL
LIN {X 0,Y 348.05,Z 382.324,A -85,B 0,C 180,E1 -13781.944,E2 -13781.944} C_VEL
LIN {X 0,Y 349.136,Z 374.063,A -85,B 0,C 180,E1 -13783.681,E2 -13783.681} C_VEL
LIN {X 0,Y 350.138,Z 365.589,A -85,B 0,C 180,E1 -13785.125,E2 -13785.125} C_VEL
LIN {X 0,Y 351.306,Z 355.116,A -85,B 0,C 180,E1 -13786.562,E2 -13786.562} C_VEL
LIN {X 0,Y 352.551,Z 343.324,A -85,B 0,C 180,E1 -13787.847,E2 -13787.847} C_VEL
LIN {X 0,Y 353.76,Z 331.453,A -85,B 0,C 180,E1 -13788.833,E2 -13788.833} C_VEL
LIN {X 0,Y 354.737,Z 319.094,A -85,B 0,C 180,E1 -13789.606,E2 -13789.606} C_VEL
LIN {X 0,Y 355.455,Z 306.383,A -85,B 0,C 180,E1 -13790.167,E2 -13790.167} C_VEL
LIN {X 0,Y 355.946,Z 293.005,A -85,B 0,C 180,E1 -13790.515,E2 -13790.515} C_VEL
LIN {X 0,Y 356.976,Z 225.143,A -85,B 0,C 180,E1 -13791.887,E2 -13791.887} C_VEL
LIN {X 0,Y 352.169,Z 198.429,A -85,B 0,C 180,E1 -13792.777,E2 -13792.777} C_VEL
LIN {X 0,Y 351.199,Z 193.386,A -85,B 0,C 180,E1 -13792.996,E2 -13792.996} C_VEL
LIN {X 0,Y 351.476,Z 188.509,A -85,B 0,C 180,E1 -13794.198,E2 -13794.198} C_VEL
LIN {X 0,Y 349.131,Z 176.266,A -85,B 0,C 180,E1 -13797.659,E2 -13797.659} C_VEL
LIN {X 0,Y 347.767,Z 170.185,A -85,B 0,C 180,E1 -13799.546,E2 -13799.546} C_VEL
LIN {X 0,Y 347.73,Z 170.162,A -85,B 0,C 180,E1 -13803.071,E2 -13803.071} C_VEL
LIN {X 0,Y 347.766,Z 170.167,A -85,B 0,C 180,E1 -13806.064,E2 -13806.064} C_VEL
LIN {X 0,Y 347.726,Z 170.15,A -85,B 0,C 180,E1 -13808.794,E2 -13808.794} C_VEL
LIN {X 0,Y 347.744,Z 170.166,A -85,B 0,C 180,E1 -13811.829,E2 -13811.829} C_VEL
LIN {X 0,Y 347.7,Z 170.176,A -85,B 0,C 180,E1 -13815.026,E2 -13815.026} C_VEL
LIN {X 0,Y 347.743,Z 170.166,A -85,B 0,C 180,E1 -13818.396,E2 -13818.396} C_VEL
LIN {X 0,Y 347.765,Z 170.142,A -85,B 0,C 180,E1 -13822.011,E2 -13822.011} C_VEL
LIN {X 0,Y 347.736,Z 170.156,A -85,B 0,C 180,E1 -13825.535,E2 -13825.535} C_VEL
LIN {X 0,Y 347.736,Z 170.169,A -85,B 0,C 180,E1 -13828.299,E2 -13828.299} C_VEL
LIN {X 0,Y 347.77,Z 170.157,A -85,B 0,C 180,E1 -13830.987,E2 -13830.987} C_VEL
LIN {X 0,Y 347.821,Z 170.157,A -85,B 0,C 180,E1 -13833.607,E2 -13833.607} C_VEL
LIN {X 0,Y 347.775,Z 170.151,A -85,B 0,C 180,E1 -13836.161,E2 -13836.161} C_VEL
LIN {X 0,Y 347.793,Z 170.159,A -85,B 0,C 180,E1 -13839.908,E2 -13839.908} C_VEL
LIN {X 0,Y 347.821,Z 170.153,A -85,B 0,C 180,E1 -13843.568,E2 -13843.568} C_VEL
LIN {X 0,Y 347.883,Z 170.142,A -85,B 0,C 180,E1 -13847.16,E2 -13847.16} C_VEL
LIN {X 0,Y 347.954,Z 170.14,A -85,B 0,C 180,E1 -13850.701,E2 -13850.701} C_VEL
LIN {X 0,Y 348.081,Z 170.122,A -85,B 0,C 180,E1 -13853.042,E2 -13853.042} C_VEL
LIN {X 0,Y 348.194,Z 170.108,A -85,B 0,C 180,E1 -13857.686,E2 -13857.686} C_VEL
LIN {X 0,Y 348.334,Z 170.094,A -85,B 0,C 180,E1 -13860,E2 -13860} C_VEL
LIN {X 0,Y 348.193,Z 170.098,A -85,B 0,C 180,E1 -13862.314,E2 -13862.314} C_VEL
LIN {X 0,Y 348.093,Z 170.119,A -85,B 0,C 180,E1 -13866.958,E2 -13866.958} C_VEL
LIN {X 0,Y 347.917,Z 170.136,A -85,B 0,C 180,E1 -13870.475,E2 -13870.475} C_VEL
LIN {X 0,Y 347.889,Z 170.145,A -85,B 0,C 180,E1 -13874.15,E2 -13874.15} C_VEL
LIN {X 0,Y 347.881,Z 170.151,A -85,B 0,C 180,E1 -13878.291,E2 -13878.291} C_VEL
LIN {X 0,Y 347.779,Z 170.154,A -85,B 0,C 180,E1 -13881.636,E2 -13881.636} C_VEL
LIN {X 0,Y 347.803,Z 170.159,A -85,B 0,C 180,E1 -13885.109,E2 -13885.109} C_VEL
LIN {X 0,Y 347.801,Z 170.151,A -85,B 0,C 180,E1 -13887.695,E2 -13887.695} C_VEL
LIN {X 0,Y 347.756,Z 170.169,A -85,B 0,C 180,E1 -13890.347,E2 -13890.347} C_VEL
LIN {X 0,Y 347.737,Z 170.133,A -85,B 0,C 180,E1 -13894.465,E2 -13894.465} C_VEL
LIN {X 0,Y 347.767,Z 170.156,A -85,B 0,C 180,E1 -13897.99,E2 -13897.99} C_VEL
LIN {X 0,Y 347.744,Z 170.153,A -85,B 0,C 180,E1 -13901.831,E2 -13901.831} C_VEL
LIN {X 0,Y 347.7,Z 170.163,A -85,B 0,C 180,E1 -13905.028,E2 -13905.028} C_VEL
LIN {X 0,Y 347.745,Z 170.159,A -85,B 0,C 180,E1 -13908.399,E2 -13908.399} C_VEL
LIN {X 0,Y 347.769,Z 170.16,A -85,B 0,C 180,E1 -13912.013,E2 -13912.013} C_VEL
LIN {X 0,Y 347.741,Z 170.155,A -85,B 0,C 180,E1 -13915.537,E2 -13915.537} C_VEL
LIN {X 0,Y 347.758,Z 170.161,A -85,B 0,C 180,E1 -13919.654,E2 -13919.654} C_VEL
LIN {X 0,Y 347.858,Z 170.375,A -85,B 0,C 180,E1 -13922.066,E2 -13922.066} C_VEL
LIN {X 0,Y 349.946,Z 180.369,A -85,B 0,C 180,E1 -13925.056,E2 -13925.056} C_VEL
LIN {X 0,Y 351.265,Z 187.6,A -85,B 0,C 180,E1 -13927.057,E2 -13927.057} C_VEL
LIN {X 0,Y 352.929,Z 194.922,A -85,B 0,C 180,E1 -13927.373,E2 -13927.373} C_VEL
LIN {X 0,Y 357.178,Z 217.471,A -85,B 0,C 180,E1 -13928.137,E2 -13928.137} C_VEL
LIN {X 0,Y 355.81,Z 295.586,A -85,B 0,C 180,E1 -13929.741,E2 -13929.741} C_VEL
LIN {X 0,Y 355.164,Z 308.615,A -85,B 0,C 180,E1 -13930.231,E2 -13930.231} C_VEL
LIN {X 0,Y 354.339,Z 320.643,A -85,B 0,C 180,E1 -13930.898,E2 -13930.898} C_VEL
LIN {X 0,Y 353.321,Z 331.998,A -85,B 0,C 180,E1 -13931.744,E2 -13931.744} C_VEL
LIN {X 0,Y 352.109,Z 343.925,A -85,B 0,C 180,E1 -13932.909,E2 -13932.909} C_VEL
LIN {X 0,Y 351.005,Z 354.552,A -85,B 0,C 180,E1 -13934.227,E2 -13934.227} C_VEL
LIN {X 0,Y 349.843,Z 364.403,A -85,B 0,C 180,E1 -13935.755,E2 -13935.755} C_VEL
LIN {X 0,Y 348.631,Z 373.34,A -85,B 0,C 180,E1 -13937.485,E2 -13937.485} C_VEL
LIN {X 0,Y 347.796,Z 380.535,A -85,B 0,C 180,E1 -13939.228,E2 -13939.228} C_VEL
LIN {X 0,Y 347.191,Z 385.389,A -85,B 0,C 180,E1 -13940.681,E2 -13940.681} C_VEL
LIN {X 0,Y 346.743,Z 390.106,A -85,B 0,C 180,E1 -13942.43,E2 -13942.43} C_VEL
LIN {X 0,Y 346.422,Z 393.718,A -85,B 0,C 180,E1 -13944.179,E2 -13944.179} C_VEL
LIN {X 0,Y 346.317,Z 395.584,A -85,B 0,C 180,E1 -13945.345,E2 -13945.345} C_VEL
LIN {X 0,Y 346.184,Z 396.989,A -85,B 0,C 180,E1 -13946.509,E2 -13946.509} C_VEL
LIN {X 0,Y 346.063,Z 398.604,A -85,B 0,C 180,E1 -13948.837,E2 -13948.837} C_VEL
LIN {X 0,Y 346.077,Z 398.837,A -85,B 0,C 180,E1 -13950.001,E2 -13950.001} C_VEL
LIN {X 0,Y 346.063,Z 398.646,A -85,B 0,C 180,E1 -13951.164,E2 -13951.164} C_VEL
LIN {X 0,Y 346.181,Z 397.086,A -85,B 0,C 180,E1 -13953.492,E2 -13953.492} C_VEL
LIN {X 0,Y 346.294,Z 395.723,A -85,B 0,C 180,E1 -13954.657,E2 -13954.657} C_VEL
LIN {X 0,Y 346.508,Z 392.921,A -85,B 0,C 180,E1 -13956.363,E2 -13956.363} C_VEL
LIN {X 0,Y 346.848,Z 388.941,A -85,B 0,C 180,E1 -13958.154,E2 -13958.154} C_VEL
LIN {X 0,Y 347.411,Z 383.906,A -85,B 0,C 180,E1 -13959.902,E2 -13959.902} C_VEL
LIN {X 0,Y 348.179,Z 377.569,A -85,B 0,C 180,E1 -13961.645,E2 -13961.645} C_VEL
LIN {X 0,Y 349.155,Z 369.639,A -85,B 0,C 180,E1 -13963.384,E2 -13963.384} C_VEL
LIN {X 0,Y 350.472,Z 359.776,A -85,B 0,C 180,E1 -13965.111,E2 -13965.111} C_VEL
LIN {X 0,Y 351.513,Z 349.43,A -85,B 0,C 180,E1 -13966.553,E2 -13966.553} C_VEL
LIN {X 0,Y 352.634,Z 339.182,A -85,B 0,C 180,E1 -13967.694,E2 -13967.694} C_VEL
LIN {X 0,Y 353.744,Z 327.971,A -85,B 0,C 180,E1 -13968.685,E2 -13968.685} C_VEL
LIN {X 0,Y 354.734,Z 315.343,A -85,B 0,C 180,E1 -13969.532,E2 -13969.532} C_VEL
LIN {X 0,Y 355.537,Z 301.77,A -85,B 0,C 180,E1 -13970.163,E2 -13970.163} C_VEL
LIN {X 0,Y 355.971,Z 289.679,A -85,B 0,C 180,E1 -13970.514,E2 -13970.514} C_VEL
LIN {X 0,Y 356.842,Z 239.985,A -85,B 0,C 180,E1 -13971.514,E2 -13971.514} C_VEL
LIN {X 0,Y 356.351,Z 234.159,A -85,B 0,C 180,E1 -13971.669,E2 -13971.669} C_VEL
LIN {X 0,Y 353.782,Z 224.837,A -85,B 0,C 180,E1 -13972.035,E2 -13972.035} C_VEL
LIN {X 0,Y 351.191,Z 217.478,A -85,B 0,C 180,E1 -13972.366,E2 -13972.366} C_VEL
LIN {X 0,Y 349.143,Z 209.93,A -85,B 0,C 180,E1 -13972.669,E2 -13972.669} C_VEL
LIN {X 0,Y 345.182,Z 190.751,A -85,B 0,C 180,E1 -13973.37,E2 -13973.37} C_VEL
LIN {X 0,Y 344.084,Z 187.538,A -85,B 0,C 180,E1 -13973.58,E2 -13973.58} C_VEL
LIN {X 0,Y 341.933,Z 176.215,A -85,B 0,C 180,E1 -13976.884,E2 -13976.884} C_VEL
LIN {X 0,Y 340.768,Z 171.082,A -85,B 0,C 180,E1 -13978.548,E2 -13978.548} C_VEL
LIN {X 0,Y 340.703,Z 171.035,A -85,B 0,C 180,E1 -13981.044,E2 -13981.044} C_VEL
LIN {X 0,Y 340.718,Z 171.029,A -85,B 0,C 180,E1 -13985.278,E2 -13985.278} C_VEL
LIN {X 0,Y 340.709,Z 171.036,A -85,B 0,C 180,E1 -13988.385,E2 -13988.385} C_VEL
LIN {X 0,Y 340.698,Z 171.039,A -85,B 0,C 180,E1 -13992.045,E2 -13992.045} C_VEL
LIN {X 0,Y 340.65,Z 171.025,A -85,B 0,C 180,E1 -13996.227,E2 -13996.227} C_VEL
LIN {X 0,Y 340.687,Z 171.045,A -85,B 0,C 180,E1 -13999.752,E2 -13999.752} C_VEL
LIN {X 0,Y 340.703,Z 171.022,A -85,B 0,C 180,E1 -14003.258,E2 -14003.258} C_VEL
LIN {X 0,Y 340.69,Z 171.014,A -85,B 0,C 180,E1 -14006.153,E2 -14006.153} C_VEL
LIN {X 0,Y 340.772,Z 171.035,A -85,B 0,C 180,E1 -14010.332,E2 -14010.332} C_VEL
LIN {X 0,Y 340.8,Z 171.023,A -85,B 0,C 180,E1 -14013.019,E2 -14013.019} C_VEL
LIN {X 0,Y 340.751,Z 171.042,A -85,B 0,C 180,E1 -14015.638,E2 -14015.638} C_VEL
LIN {X 0,Y 340.73,Z 171.035,A -85,B 0,C 180,E1 -14019.473,E2 -14019.473} C_VEL
LIN {X 0,Y 340.854,Z 171.024,A -85,B 0,C 180,E1 -14021.984,E2 -14021.984} C_VEL
LIN {X 0,Y 340.865,Z 171.017,A -85,B 0,C 180,E1 -14025.705,E2 -14025.705} C_VEL
LIN {X 0,Y 340.866,Z 171.019,A -85,B 0,C 180,E1 -14029.306,E2 -14029.306} C_VEL
LIN {X 0,Y 341.069,Z 170.993,A -85,B 0,C 180,E1 -14032.898,E2 -14032.898} C_VEL
LIN {X 0,Y 341.16,Z 170.973,A -85,B 0,C 180,E1 -14037.639,E2 -14037.639} C_VEL
LIN {X 0,Y 341.27,Z 170.974,A -85,B 0,C 180,E1 -14040,E2 -14040} C_VEL
LIN {X 0,Y 341.161,Z 170.984,A -85,B 0,C 180,E1 -14042.361,E2 -14042.361} C_VEL
LIN {X 0,Y 341.039,Z 171,A -85,B 0,C 180,E1 -14047.103,E2 -14047.103} C_VEL
LIN {X 0,Y 340.842,Z 171.017,A -85,B 0,C 180,E1 -14050.695,E2 -14050.695} C_VEL
LIN {X 0,Y 340.859,Z 171.024,A -85,B 0,C 180,E1 -14054.325,E2 -14054.325} C_VEL
LIN {X 0,Y 340.782,Z 171.023,A -85,B 0,C 180,E1 -14058.441,E2 -14058.441} C_VEL
LIN {X 0,Y 340.714,Z 171.041,A -85,B 0,C 180,E1 -14061.842,E2 -14061.842} C_VEL
LIN {X 0,Y 340.768,Z 171.037,A -85,B 0,C 180,E1 -14065.665,E2 -14065.665} C_VEL
LIN {X 0,Y 340.725,Z 171.038,A -85,B 0,C 180,E1 -14068.321,E2 -14068.321} C_VEL
LIN {X 0,Y 340.694,Z 171.045,A -85,B 0,C 180,E1 -14071.045,E2 -14071.045} C_VEL
LIN {X 0,Y 340.715,Z 171.016,A -85,B 0,C 180,E1 -14075.279,E2 -14075.279} C_VEL
LIN {X 0,Y 340.707,Z 171.028,A -85,B 0,C 180,E1 -14078.386,E2 -14078.386} C_VEL
LIN {X 0,Y 340.696,Z 171.042,A -85,B 0,C 180,E1 -14082.046,E2 -14082.046} C_VEL
LIN {X 0,Y 340.65,Z 171.05,A -85,B 0,C 180,E1 -14086.228,E2 -14086.228} C_VEL
LIN {X 0,Y 340.673,Z 171.045,A -85,B 0,C 180,E1 -14089.756,E2 -14089.756} C_VEL
LIN {X 0,Y 340.702,Z 171.041,A -85,B 0,C 180,E1 -14093.258,E2 -14093.258} C_VEL
LIN {X 0,Y 340.692,Z 171.034,A -85,B 0,C 180,E1 -14096.154,E2 -14096.154} C_VEL
LIN {X 0,Y 340.753,Z 171.248,A -85,B 0,C 180,E1 -14100.155,E2 -14100.155} C_VEL
LIN {X 0,Y 343.181,Z 182.442,A -85,B 0,C 180,E1 -14103.523,E2 -14103.523} C_VEL
LIN {X 0,Y 344.63,Z 190.894,A -85,B 0,C 180,E1 -14105.93,E2 -14105.93} C_VEL
LIN {X 0,Y 344.497,Z 193.555,A -85,B 0,C 180,E1 -14106.531,E2 -14106.531} C_VEL
LIN {X 0,Y 349.473,Z 220.273,A -85,B 0,C 180,E1 -14107.496,E2 -14107.496} C_VEL
LIN {X 0,Y 350.52,Z 226.615,A -85,B 0,C 180,E1 -14107.704,E2 -14107.704} C_VEL
LIN {X 0,Y 349.13,Z 301.206,A -85,B 0,C 180,E1 -14109.258,E2 -14109.258} C_VEL
LIN {X 0,Y 348.392,Z 314.389,A -85,B 0,C 180,E1 -14109.752,E2 -14109.752} C_VEL
LIN {X 0,Y 347.43,Z 326.498,A -85,B 0,C 180,E1 -14110.425,E2 -14110.425} C_VEL
LIN {X 0,Y 346.357,Z 338.718,A -85,B 0,C 180,E1 -14111.362,E2 -14111.362} C_VEL
LIN {X 0,Y 345.091,Z 350.28,A -85,B 0,C 180,E1 -14112.519,E2 -14112.519} C_VEL
LIN {X 0,Y 343.849,Z 360.988,A -85,B 0,C 180,E1 -14113.873,E2 -14113.873} C_VEL
LIN {X 0,Y 342.895,Z 369.198,A -85,B 0,C 180,E1 -14115.155,E2 -14115.155} C_VEL
LIN {X 0,Y 341.849,Z 377.047,A -85,B 0,C 180,E1 -14116.627,E2 -14116.627} C_VEL
LIN {X 0,Y 340.799,Z 384.709,A -85,B 0,C 180,E1 -14118.4,E2 -14118.4} C_VEL
LIN {X 0,Y 339.947,Z 391.774,A -85,B 0,C 180,E1 -14120.48,E2 -14120.48} C_VEL
LIN {X 0,Y 339.471,Z 396.472,A -85,B 0,C 180,E1 -14122.266,E2 -14122.266} C_VEL
LIN {X 0,Y 339.21,Z 400.061,A -85,B 0,C 180,E1 -14124.053,E2 -14124.053} C_VEL
LIN {X 0,Y 339.124,Z 401.912,A -85,B 0,C 180,E1 -14125.245,E2 -14125.245} C_VEL
LIN {X 0,Y 339.065,Z 403.299,A -85,B 0,C 180,E1 -14126.434,E2 -14126.434} C_VEL
LIN {X 0,Y 338.957,Z 404.892,A -85,B 0,C 180,E1 -14128.811,E2 -14128.811} C_VEL
LIN {X 0,Y 338.978,Z 405.105,A -85,B 0,C 180,E1 -14129.999,E2 -14129.999} C_VEL
LIN {X 0,Y 338.956,Z 404.886,A -85,B 0,C 180,E1 -14131.188,E2 -14131.188} C_VEL
LIN {X 0,Y 339.065,Z 403.288,A -85,B 0,C 180,E1 -14133.565,E2 -14133.565} C_VEL
LIN {X 0,Y 339.123,Z 401.895,A -85,B 0,C 180,E1 -14134.754,E2 -14134.754} C_VEL
LIN {X 0,Y 339.299,Z 398.97,A -85,B 0,C 180,E1 -14136.54,E2 -14136.54} C_VEL
LIN {X 0,Y 339.612,Z 395.007,A -85,B 0,C 180,E1 -14138.328,E2 -14138.328} C_VEL
LIN {X 0,Y 340.283,Z 388.915,A -85,B 0,C 180,E1 -14140.411,E2 -14140.411} C_VEL
LIN {X 0,Y 341.09,Z 382.257,A -85,B 0,C 180,E1 -14142.192,E2 -14142.192} C_VEL
LIN {X 0,Y 342.231,Z 373.995,A -85,B 0,C 180,E1 -14143.962,E2 -14143.962} C_VEL
LIN {X 0,Y 343.415,Z 364.335,A -85,B 0,C 180,E1 -14145.614,E2 -14145.614} C_VEL
LIN {X 0,Y 344.617,Z 353.873,A -85,B 0,C 180,E1 -14147.046,E2 -14147.046} C_VEL
LIN {X 0,Y 345.795,Z 343.255,A -85,B 0,C 180,E1 -14148.208,E2 -14148.208} C_VEL
LIN {X 0,Y 347.04,Z 331.382,A -85,B 0,C 180,E1 -14149.212,E2 -14149.212} C_VEL
LIN {X 0,Y 348.046,Z 319.021,A -85,B 0,C 180,E1 -14149.999,E2 -14149.999} C_VEL
LIN {X 0,Y 348.792,Z 306.307,A -85,B 0,C 180,E1 -14150.569,E2 -14150.569} C_VEL
LIN {X 0,Y 349.303,Z 292.92,A -85,B 0,C 180,E1 -14150.923,E2 -14150.923} C_VEL
LIN {X 0,Y 350.511,Z 227.02,A -85,B 0,C 180,E1 -14152.269,E2 -14152.269} C_VEL
LIN {X 0,Y 345.983,Z 201.315,A -85,B 0,C 180,E1 -14153.142,E2 -14153.142} C_VEL
LIN {X 0,Y 344.459,Z 193.388,A -85,B 0,C 180,E1 -14153.465,E2 -14153.465} C_VEL
LIN {X 0,Y 344.494,Z 189.63,A -85,B 0,C 180,E1 -14154.4,E2 -14154.4} C_VEL
LIN {X 0,Y 342.489,Z 179.088,A -85,B 0,C 180,E1 -14157.438,E2 -14157.438} C_VEL
LIN {X 0,Y 340.713,Z 171.096,A -85,B 0,C 180,E1 -14159.915,E2 -14159.915} C_VEL
LIN {X 0,Y 340.689,Z 171.034,A -85,B 0,C 180,E1 -14163.845,E2 -14163.845} C_VEL
LIN {X 0,Y 340.698,Z 171.04,A -85,B 0,C 180,E1 -14166.741,E2 -14166.741} C_VEL
LIN {X 0,Y 340.671,Z 171.046,A -85,B 0,C 180,E1 -14170.243,E2 -14170.243} C_VEL
LIN {X 0,Y 340.646,Z 171.051,A -85,B 0,C 180,E1 -14173.772,E2 -14173.772} C_VEL
LIN {X 0,Y 340.692,Z 171.043,A -85,B 0,C 180,E1 -14177.954,E2 -14177.954} C_VEL
LIN {X 0,Y 340.725,Z 171.022,A -85,B 0,C 180,E1 -14181.771,E2 -14181.771} C_VEL
LIN {X 0,Y 340.715,Z 171.031,A -85,B 0,C 180,E1 -14185.595,E2 -14185.595} C_VEL
LIN {X 0,Y 340.689,Z 171.045,A -85,B 0,C 180,E1 -14188.954,E2 -14188.954} C_VEL
LIN {X 0,Y 340.767,Z 171.035,A -85,B 0,C 180,E1 -14192.474,E2 -14192.474} C_VEL
LIN {X 0,Y 340.745,Z 171.027,A -85,B 0,C 180,E1 -14195.637,E2 -14195.637} C_VEL
LIN {X 0,Y 340.722,Z 171.041,A -85,B 0,C 180,E1 -14199.473,E2 -14199.473} C_VEL
LIN {X 0,Y 340.782,Z 171.021,A -85,B 0,C 180,E1 -14201.98,E2 -14201.98} C_VEL
LIN {X 0,Y 340.859,Z 171.024,A -85,B 0,C 180,E1 -14205.705,E2 -14205.705} C_VEL
LIN {X 0,Y 340.863,Z 171.015,A -85,B 0,C 180,E1 -14209.306,E2 -14209.306} C_VEL
LIN {X 0,Y 341.049,Z 170.999,A -85,B 0,C 180,E1 -14212.898,E2 -14212.898} C_VEL
LIN {X 0,Y 341.156,Z 170.985,A -85,B 0,C 180,E1 -14217.639,E2 -14217.639} C_VEL
LIN {X 0,Y 341.284,Z 170.972,A -85,B 0,C 180,E1 -14220,E2 -14220} C_VEL
LIN {X 0,Y 341.155,Z 170.974,A -85,B 0,C 180,E1 -14222.361,E2 -14222.361} C_VEL
LIN {X 0,Y 341.063,Z 170.994,A -85,B 0,C 180,E1 -14227.102,E2 -14227.102} C_VEL
LIN {X 0,Y 340.86,Z 171.018,A -85,B 0,C 180,E1 -14230.694,E2 -14230.694} C_VEL
LIN {X 0,Y 340.853,Z 171.019,A -85,B 0,C 180,E1 -14234.325,E2 -14234.325} C_VEL
LIN {X 0,Y 340.828,Z 171.032,A -85,B 0,C 180,E1 -14238.467,E2 -14238.467} C_VEL
LIN {X 0,Y 340.745,Z 171.029,A -85,B 0,C 180,E1 -14241.858,E2 -14241.858} C_VEL
LIN {X 0,Y 340.763,Z 171.038,A -85,B 0,C 180,E1 -14245.665,E2 -14245.665} C_VEL
LIN {X 0,Y 340.732,Z 171.033,A -85,B 0,C 180,E1 -14248.321,E2 -14248.321} C_VEL
LIN {X 0,Y 340.696,Z 171.044,A -85,B 0,C 180,E1 -14251.045,E2 -14251.045} C_VEL
LIN {X 0,Y 340.71,Z 171.004,A -85,B 0,C 180,E1 -14255.28,E2 -14255.28} C_VEL
LIN {X 0,Y 340.703,Z 171.042,A -85,B 0,C 180,E1 -14258.387,E2 -14258.387} C_VEL
LIN {X 0,Y 340.693,Z 171.028,A -85,B 0,C 180,E1 -14262.047,E2 -14262.047} C_VEL
LIN {X 0,Y 340.647,Z 171.053,A -85,B 0,C 180,E1 -14266.228,E2 -14266.228} C_VEL
LIN {X 0,Y 340.683,Z 171.026,A -85,B 0,C 180,E1 -14269.754,E2 -14269.754} C_VEL
LIN {X 0,Y 340.701,Z 171.047,A -85,B 0,C 180,E1 -14273.26,E2 -14273.26} C_VEL
LIN {X 0,Y 340.69,Z 171.038,A -85,B 0,C 180,E1 -14276.155,E2 -14276.155} C_VEL
LIN {X 0,Y 340.783,Z 171.038,A -85,B 0,C 180,E1 -14280.335,E2 -14280.335} C_VEL
LIN {X 0,Y 340.778,Z 171.129,A -85,B 0,C 180,E1 -14281.601,E2 -14281.601} C_VEL
LIN {X 0,Y 342.981,Z 181.592,A -85,B 0,C 180,E1 -14284.839,E2 -14284.839} C_VEL
LIN {X 0,Y 344.105,Z 187.642,A -85,B 0,C 180,E1 -14286.546,E2 -14286.546} C_VEL
LIN {X 0,Y 345.655,Z 192.728,A -85,B 0,C 180,E1 -14286.818,E2 -14286.818} C_VEL
LIN {X 0,Y 350.567,Z 218.013,A -85,B 0,C 180,E1 -14287.713,E2 -14287.713} C_VEL
LIN {X 0,Y 349.174,Z 295.667,A -85,B 0,C 180,E1 -14289.339,E2 -14289.339} C_VEL
LIN {X 0,Y 348.473,Z 308.691,A -85,B 0,C 180,E1 -14289.835,E2 -14289.835} C_VEL
LIN {X 0,Y 347.647,Z 320.715,A -85,B 0,C 180,E1 -14290.516,E2 -14290.516} C_VEL
LIN {X 0,Y 346.606,Z 332.069,A -85,B 0,C 180,E1 -14291.377,E2 -14291.377} C_VEL
LIN {X 0,Y 345.355,Z 343.737,A -85,B 0,C 180,E1 -14292.534,E2 -14292.534} C_VEL
LIN {X 0,Y 344.246,Z 353.964,A -85,B 0,C 180,E1 -14293.815,E2 -14293.815} C_VEL
LIN {X 0,Y 343.208,Z 362.773,A -85,B 0,C 180,E1 -14295.17,E2 -14295.17} C_VEL
LIN {X 0,Y 342.095,Z 370.663,A -85,B 0,C 180,E1 -14296.638,E2 -14296.638} C_VEL
LIN {X 0,Y 341.102,Z 378.375,A -85,B 0,C 180,E1 -14298.412,E2 -14298.412} C_VEL
LIN {X 0,Y 340.19,Z 385.455,A -85,B 0,C 180,E1 -14300.488,E2 -14300.488} C_VEL
LIN {X 0,Y 339.686,Z 390.172,A -85,B 0,C 180,E1 -14302.272,E2 -14302.272} C_VEL
LIN {X 0,Y 339.347,Z 393.784,A -85,B 0,C 180,E1 -14304.057,E2 -14304.057} C_VEL
LIN {X 0,Y 339.238,Z 395.649,A -85,B 0,C 180,E1 -14305.247,E2 -14305.247} C_VEL
LIN {X 0,Y 339.113,Z 397.054,A -85,B 0,C 180,E1 -14306.436,E2 -14306.436} C_VEL
LIN {X 0,Y 338.969,Z 398.669,A -85,B 0,C 180,E1 -14308.813,E2 -14308.813} C_VEL
LIN {X 0,Y 338.98,Z 398.902,A -85,B 0,C 180,E1 -14310.001,E2 -14310.001} C_VEL
LIN {X 0,Y 338.969,Z 398.711,A -85,B 0,C 180,E1 -14311.189,E2 -14311.189} C_VEL
LIN {X 0,Y 339.109,Z 397.151,A -85,B 0,C 180,E1 -14313.565,E2 -14313.565} C_VEL
LIN {X 0,Y 339.217,Z 395.788,A -85,B 0,C 180,E1 -14314.754,E2 -14314.754} C_VEL
LIN {X 0,Y 339.416,Z 393.279,A -85,B 0,C 180,E1 -14316.331,E2 -14316.331} C_VEL
LIN {X 0,Y 339.803,Z 389.004,A -85,B 0,C 180,E1 -14318.325,E2 -14318.325} C_VEL
LIN {X 0,Y 340.4,Z 383.969,A -85,B 0,C 180,E1 -14320.108,E2 -14320.108} C_VEL
LIN {X 0,Y 341.188,Z 377.632,A -85,B 0,C 180,E1 -14321.887,E2 -14321.887} C_VEL
LIN {X 0,Y 342.252,Z 369.701,A -85,B 0,C 180,E1 -14323.659,E2 -14323.659} C_VEL
LIN {X 0,Y 343.63,Z 359.838,A -85,B 0,C 180,E1 -14325.419,E2 -14325.419} C_VEL
LIN {X 0,Y 344.559,Z 350.662,A -85,B 0,C 180,E1 -14326.745,E2 -14326.745} C_VEL
LIN {X 0,Y 345.866,Z 339.242,A -85,B 0,C 180,E1 -14328.052,E2 -14328.052} C_VEL
LIN {X 0,Y 347.023,Z 328.03,A -85,B 0,C 180,E1 -14329.061,E2 -14329.061} C_VEL
LIN {X 0,Y 348.055,Z 315.399,A -85,B 0,C 180,E1 -14329.922,E2 -14329.922} C_VEL
LIN {X 0,Y 348.903,Z 301.822,A -85,B 0,C 180,E1 -14330.564,E2 -14330.564} C_VEL
LIN {X 0,Y 349.352,Z 289.723,A -85,B 0,C 180,E1 -14330.921,E2 -14330.921} C_VEL
LIN {X 0,Y 350.535,Z 217.825,A -85,B 0,C 180,E1 -14332.402,E2 -14332.402} C_VEL
LIN {X 0,Y 349.143,Z 209.93,A -85,B 0,C 180,E1 -14332.669,E2 -14332.669} C_VEL
LIN {X 0,Y 347.856,Z 206.335,A -85,B 0,C 180,E1 -14332.837,E2 -14332.837} C_VEL
LIN {X 0,Y 344.246,Z 201.173,A -85,B 0,C 180,E1 -14333.205,E2 -14333.205} C_VEL
LIN {X 0,Y 339.733,Z 195.015,A -85,B 0,C 180,E1 -14333.672,E2 -14333.672} C_VEL
LIN {X 0,Y 338.699,Z 192.657,A -85,B 0,C 180,E1 -14333.802,E2 -14333.802} C_VEL
LIN {X 0,Y 336.952,Z 187.811,A -85,B 0,C 180,E1 -14334.083,E2 -14334.083} C_VEL
LIN {X 0,Y 335.806,Z 181.667,A -85,B 0,C 180,E1 -14335.85,E2 -14335.85} C_VEL
LIN {X 0,Y 333.772,Z 172.226,A -85,B 0,C 180,E1 -14338.812,E2 -14338.812} C_VEL
LIN {X 0,Y 333.741,Z 171.91,A -85,B 0,C 180,E1 -14339.314,E2 -14339.314} C_VEL
LIN {X 0,Y 333.637,Z 171.926,A -85,B 0,C 180,E1 -14343.208,E2 -14343.208} C_VEL
LIN {X 0,Y 333.676,Z 171.913,A -85,B 0,C 180,E1 -14346.139,E2 -14346.139} C_VEL
LIN {X 0,Y 333.646,Z 171.905,A -85,B 0,C 180,E1 -14349.192,E2 -14349.192} C_VEL
LIN {X 0,Y 333.632,Z 171.925,A -85,B 0,C 180,E1 -14352.499,E2 -14352.499} C_VEL
LIN {X 0,Y 333.594,Z 171.906,A -85,B 0,C 180,E1 -14355.954,E2 -14355.954} C_VEL
LIN {X 0,Y 333.646,Z 171.919,A -85,B 0,C 180,E1 -14359.315,E2 -14359.315} C_VEL
LIN {X 0,Y 333.663,Z 171.9,A -85,B 0,C 180,E1 -14363.167,E2 -14363.167} C_VEL
LIN {X 0,Y 333.671,Z 171.879,A -85,B 0,C 180,E1 -14365.341,E2 -14365.341} C_VEL
LIN {X 0,Y 333.7,Z 171.919,A -85,B 0,C 180,E1 -14369.71,E2 -14369.71} C_VEL
LIN {X 0,Y 333.739,Z 171.902,A -85,B 0,C 180,E1 -14372.401,E2 -14372.401} C_VEL
LIN {X 0,Y 333.722,Z 171.914,A -85,B 0,C 180,E1 -14375.09,E2 -14375.09} C_VEL
LIN {X 0,Y 333.669,Z 171.912,A -85,B 0,C 180,E1 -14379.018,E2 -14379.018} C_VEL
LIN {X 0,Y 333.79,Z 171.909,A -85,B 0,C 180,E1 -14381.589,E2 -14381.589} C_VEL
LIN {X 0,Y 333.804,Z 171.894,A -85,B 0,C 180,E1 -14385.576,E2 -14385.576} C_VEL
LIN {X 0,Y 333.829,Z 171.897,A -85,B 0,C 180,E1 -14389.078,E2 -14389.078} C_VEL
LIN {X 0,Y 334.019,Z 171.871,A -85,B 0,C 180,E1 -14392.747,E2 -14392.747} C_VEL
LIN {X 0,Y 333.8,Z 171.904,A -85,B 0,C 180,E1 -14395.169,E2 -14395.169} C_VEL
LIN {X 0,Y 334.098,Z 171.852,A -85,B 0,C 180,E1 -14397.589,E2 -14397.589} C_VEL
LIN {X 0,Y 334.221,Z 171.852,A -85,B 0,C 180,E1 -14400,E2 -14400} C_VEL
LIN {X 0,Y 334.098,Z 171.864,A -85,B 0,C 180,E1 -14402.411,E2 -14402.411} C_VEL
LIN {X 0,Y 334.001,Z 171.874,A -85,B 0,C 180,E1 -14406.039,E2 -14406.039} C_VEL
LIN {X 0,Y 333.815,Z 171.896,A -85,B 0,C 180,E1 -14409.696,E2 -14409.696} C_VEL
LIN {X 0,Y 333.788,Z 171.903,A -85,B 0,C 180,E1 -14413.392,E2 -14413.392} C_VEL
LIN {X 0,Y 333.714,Z 171.905,A -85,B 0,C 180,E1 -14417.148,E2 -14417.148} C_VEL
LIN {X 0,Y 333.712,Z 171.915,A -85,B 0,C 180,E1 -14419.692,E2 -14419.692} C_VEL
LIN {X 0,Y 333.665,Z 171.91,A -85,B 0,C 180,E1 -14423.591,E2 -14423.591} C_VEL
LIN {X 0,Y 333.731,Z 171.912,A -85,B 0,C 180,E1 -14426.247,E2 -14426.247} C_VEL
LIN {X 0,Y 333.687,Z 171.911,A -85,B 0,C 180,E1 -14428.974,E2 -14428.974} C_VEL
LIN {X 0,Y 333.64,Z 171.926,A -85,B 0,C 180,E1 -14432.587,E2 -14432.587} C_VEL
LIN {X 0,Y 333.673,Z 171.885,A -85,B 0,C 180,E1 -14436.139,E2 -14436.139} C_VEL
LIN {X 0,Y 333.644,Z 171.915,A -85,B 0,C 180,E1 -14439.193,E2 -14439.193} C_VEL
LIN {X 0,Y 333.63,Z 171.92,A -85,B 0,C 180,E1 -14442.5,E2 -14442.5} C_VEL
LIN {X 0,Y 333.594,Z 171.929,A -85,B 0,C 180,E1 -14445.955,E2 -14445.955} C_VEL
LIN {X 0,Y 333.641,Z 171.923,A -85,B 0,C 180,E1 -14449.317,E2 -14449.317} C_VEL
LIN {X 0,Y 333.662,Z 171.915,A -85,B 0,C 180,E1 -14453.169,E2 -14453.169} C_VEL
LIN {X 0,Y 333.674,Z 171.911,A -85,B 0,C 180,E1 -14455.342,E2 -14455.342} C_VEL
LIN {X 0,Y 333.667,Z 171.917,A -85,B 0,C 180,E1 -14459.548,E2 -14459.548} C_VEL
LIN {X 0,Y 333.688,Z 172.082,A -85,B 0,C 180,E1 -14459.715,E2 -14459.715} C_VEL
LIN {X 0,Y 335.973,Z 182.47,A -85,B 0,C 180,E1 -14462.937,E2 -14462.937} C_VEL
LIN {X 0,Y 337.671,Z 191.883,A -85,B 0,C 180,E1 -14465.691,E2 -14465.691} C_VEL
LIN {X 0,Y 337.673,Z 193.327,A -85,B 0,C 180,E1 -14466.014,E2 -14466.014} C_VEL
LIN {X 0,Y 340.553,Z 208.049,A -85,B 0,C 180,E1 -14466.599,E2 -14466.599} C_VEL
LIN {X 0,Y 343.985,Z 227.962,A -85,B 0,C 180,E1 -14467.288,E2 -14467.288} C_VEL
LIN {X 0,Y 342.499,Z 301.154,A -85,B 0,C 180,E1 -14468.837,E2 -14468.837} C_VEL
LIN {X 0,Y 341.73,Z 314.333,A -85,B 0,C 180,E1 -14469.339,E2 -14469.339} C_VEL
LIN {X 0,Y 340.758,Z 326.44,A -85,B 0,C 180,E1 -14470.026,E2 -14470.026} C_VEL
LIN {X 0,Y 339.633,Z 338.658,A -85,B 0,C 180,E1 -14470.979,E2 -14470.979} C_VEL
LIN {X 0,Y 338.32,Z 350.219,A -85,B 0,C 180,E1 -14472.157,E2 -14472.157} C_VEL
LIN {X 0,Y 336.986,Z 361.053,A -85,B 0,C 180,E1 -14473.554,E2 -14473.554} C_VEL
LIN {X 0,Y 335.793,Z 370.806,A -85,B 0,C 180,E1 -14475.144,E2 -14475.144} C_VEL
LIN {X 0,Y 334.484,Z 379.711,A -85,B 0,C 180,E1 -14476.946,E2 -14476.946} C_VEL
LIN {X 0,Y 333.572,Z 386.875,A -85,B 0,C 180,E1 -14478.762,E2 -14478.762} C_VEL
LIN {X 0,Y 332.741,Z 393.398,A -85,B 0,C 180,E1 -14480.885,E2 -14480.885} C_VEL
LIN {X 0,Y 332.291,Z 397.713,A -85,B 0,C 180,E1 -14482.709,E2 -14482.709} C_VEL
LIN {X 0,Y 332.136,Z 400.127,A -85,B 0,C 180,E1 -14484.001,E2 -14484.001} C_VEL
LIN {X 0,Y 332.031,Z 401.847,A -85,B 0,C 180,E1 -14485.143,E2 -14485.143} C_VEL
LIN {X 0,Y 331.973,Z 403.234,A -85,B 0,C 180,E1 -14486.358,E2 -14486.358} C_VEL
LIN {X 0,Y 331.865,Z 404.827,A -85,B 0,C 180,E1 -14488.786,E2 -14488.786} C_VEL
LIN {X 0,Y 331.884,Z 405.04,A -85,B 0,C 180,E1 -14489.999,E2 -14489.999} C_VEL
LIN {X 0,Y 331.865,Z 404.821,A -85,B 0,C 180,E1 -14491.213,E2 -14491.213} C_VEL
LIN {X 0,Y 331.972,Z 403.222,A -85,B 0,C 180,E1 -14493.641,E2 -14493.641} C_VEL
LIN {X 0,Y 332.031,Z 401.829,A -85,B 0,C 180,E1 -14494.856,E2 -14494.856} C_VEL
LIN {X 0,Y 332.244,Z 398.903,A -85,B 0,C 180,E1 -14496.68,E2 -14496.68} C_VEL
LIN {X 0,Y 332.575,Z 394.941,A -85,B 0,C 180,E1 -14498.506,E2 -14498.506} C_VEL
LIN {X 0,Y 333.273,Z 388.848,A -85,B 0,C 180,E1 -14500.632,E2 -14500.632} C_VEL
LIN {X 0,Y 334.128,Z 382.19,A -85,B 0,C 180,E1 -14502.45,E2 -14502.45} C_VEL
LIN {X 0,Y 335.329,Z 373.928,A -85,B 0,C 180,E1 -14504.256,E2 -14504.256} C_VEL
LIN {X 0,Y 336.415,Z 365.454,A -85,B 0,C 180,E1 -14505.757,E2 -14505.757} C_VEL
LIN {X 0,Y 337.665,Z 354.979,A -85,B 0,C 180,E1 -14507.252,E2 -14507.252} C_VEL
LIN {X 0,Y 339.049,Z 343.186,A -85,B 0,C 180,E1 -14508.583,E2 -14508.583} C_VEL
LIN {X 0,Y 340.35,Z 331.311,A -85,B 0,C 180,E1 -14509.605,E2 -14509.605} C_VEL
LIN {X 0,Y 341.395,Z 318.949,A -85,B 0,C 180,E1 -14510.405,E2 -14510.405} C_VEL
LIN {X 0,Y 342.169,Z 306.231,A -85,B 0,C 180,E1 -14510.986,E2 -14510.986} C_VEL
LIN {X 0,Y 342.695,Z 292.834,A -85,B 0,C 180,E1 -14511.346,E2 -14511.346} C_VEL
LIN {X 0,Y 343.832,Z 226.93,A -85,B 0,C 180,E1 -14512.726,E2 -14512.726} C_VEL
LIN {X 0,Y 339.208,Z 201.226,A -85,B 0,C 180,E1 -14513.632,E2 -14513.632} C_VEL
LIN {X 0,Y 337.655,Z 193.268,A -85,B 0,C 180,E1 -14513.972,E2 -14513.972} C_VEL
LIN {X 0,Y 337.539,Z 190.751,A -85,B 0,C 180,E1 -14514.608,E2 -14514.608} C_VEL
LIN {X 0,Y 335.111,Z 178.445,A -85,B 0,C 180,E1 -14518.257,E2 -14518.257} C_VEL
LIN {X 0,Y 333.679,Z 171.966,A -85,B 0,C 180,E1 -14520.338,E2 -14520.338} C_VEL
LIN {X 0,Y 333.633,Z 171.915,A -85,B 0,C 180,E1 -14523.207,E2 -14523.207} C_VEL
LIN {X 0,Y 333.671,Z 171.922,A -85,B 0,C 180,E1 -14526.138,E2 -14526.138} C_VEL
LIN {X 0,Y 333.628,Z 171.908,A -85,B 0,C 180,E1 -14529.193,E2 -14529.193} C_VEL
LIN {X 0,Y 333.626,Z 171.922,A -85,B 0,C 180,E1 -14532.499,E2 -14532.499} C_VEL
LIN {X 0,Y 333.59,Z 171.926,A -85,B 0,C 180,E1 -14535.954,E2 -14535.954} C_VEL
LIN {X 0,Y 333.641,Z 171.925,A -85,B 0,C 180,E1 -14539.314,E2 -14539.314} C_VEL
LIN {X 0,Y 333.657,Z 171.886,A -85,B 0,C 180,E1 -14543.167,E2 -14543.167} C_VEL
LIN {X 0,Y 333.666,Z 171.903,A -85,B 0,C 180,E1 -14545.34,E2 -14545.34} C_VEL
LIN {X 0,Y 333.682,Z 171.912,A -85,B 0,C 180,E1 -14549.636,E2 -14549.636} C_VEL
LIN {X 0,Y 333.731,Z 171.911,A -85,B 0,C 180,E1 -14552.4,E2 -14552.4} C_VEL
LIN {X 0,Y 333.716,Z 171.906,A -85,B 0,C 180,E1 -14555.09,E2 -14555.09} C_VEL
LIN {X 0,Y 333.662,Z 171.923,A -85,B 0,C 180,E1 -14559.018,E2 -14559.018} C_VEL
LIN {X 0,Y 333.731,Z 171.9,A -85,B 0,C 180,E1 -14561.586,E2 -14561.586} C_VEL
LIN {X 0,Y 333.798,Z 171.903,A -85,B 0,C 180,E1 -14565.576,E2 -14565.576} C_VEL
LIN {X 0,Y 333.826,Z 171.889,A -85,B 0,C 180,E1 -14569.078,E2 -14569.078} C_VEL
LIN {X 0,Y 334.001,Z 171.878,A -85,B 0,C 180,E1 -14572.747,E2 -14572.747} C_VEL
LIN {X 0,Y 333.794,Z 171.888,A -85,B 0,C 180,E1 -14575.169,E2 -14575.169} C_VEL
LIN {X 0,Y 334.093,Z 171.865,A -85,B 0,C 180,E1 -14577.589,E2 -14577.589} C_VEL
LIN {X 0,Y 334.235,Z 171.85,A -85,B 0,C 180,E1 -14580,E2 -14580} C_VEL
LIN {X 0,Y 334.092,Z 171.853,A -85,B 0,C 180,E1 -14582.411,E2 -14582.411} C_VEL
LIN {X 0,Y 334.013,Z 171.872,A -85,B 0,C 180,E1 -14587.253,E2 -14587.253} C_VEL
LIN {X 0,Y 333.823,Z 171.898,A -85,B 0,C 180,E1 -14590.922,E2 -14590.922} C_VEL
LIN {X 0,Y 333.799,Z 171.894,A -85,B 0,C 180,E1 -14594.635,E2 -14594.635} C_VEL
LIN {X 0,Y 333.787,Z 171.907,A -85,B 0,C 180,E1 -14598.656,E2 -14598.656} C_VEL
LIN {X 0,Y 333.683,Z 171.908,A -85,B 0,C 180,E1 -14602.279,E2 -14602.279} C_VEL
LIN {X 0,Y 333.726,Z 171.91,A -85,B 0,C 180,E1 -14606.247,E2 -14606.247} C_VEL
LIN {X 0,Y 333.702,Z 171.913,A -85,B 0,C 180,E1 -14608.973,E2 -14608.973} C_VEL
LIN {X 0,Y 333.636,Z 171.913,A -85,B 0,C 180,E1 -14612.588,E2 -14612.588} C_VEL
LIN {X 0,Y 333.669,Z 171.885,A -85,B 0,C 180,E1 -14616.14,E2 -14616.14} C_VEL
LIN {X 0,Y 333.64,Z 171.924,A -85,B 0,C 180,E1 -14619.193,E2 -14619.193} C_VEL
LIN {X 0,Y 333.626,Z 171.904,A -85,B 0,C 180,E1 -14622.501,E2 -14622.501} C_VEL
LIN {X 0,Y 333.591,Z 171.927,A -85,B 0,C 180,E1 -14625.956,E2 -14625.956} C_VEL
LIN {X 0,Y 333.643,Z 171.905,A -85,B 0,C 180,E1 -14629.317,E2 -14629.317} C_VEL
LIN {X 0,Y 333.661,Z 171.924,A -85,B 0,C 180,E1 -14633.169,E2 -14633.169} C_VEL
LIN {X 0,Y 333.671,Z 171.906,A -85,B 0,C 180,E1 -14635.343,E2 -14635.343} C_VEL
LIN {X 0,Y 333.702,Z 171.912,A -85,B 0,C 180,E1 -14639.711,E2 -14639.711} C_VEL
LIN {X 0,Y 333.742,Z 172.103,A -85,B 0,C 180,E1 -14641.247,E2 -14641.247} C_VEL
LIN {X 0,Y 335.733,Z 181.384,A -85,B 0,C 180,E1 -14644.176,E2 -14644.176} C_VEL
LIN {X 0,Y 336.932,Z 187.703,A -85,B 0,C 180,E1 -14646.014,E2 -14646.014} C_VEL
LIN {X 0,Y 339.186,Z 194.211,A -85,B 0,C 180,E1 -14646.381,E2 -14646.381} C_VEL
LIN {X 0,Y 343.885,Z 218.258,A -85,B 0,C 180,E1 -14647.259,E2 -14647.259} C_VEL
LIN {X 0,Y 343.448,Z 252.526,A -85,B 0,C 180,E1 -14647.988,E2 -14647.988} C_VEL
LIN {X 0,Y 342.556,Z 295.747,A -85,B 0,C 180,E1 -14648.921,E2 -14648.921} C_VEL
LIN {X 0,Y 341.817,Z 308.766,A -85,B 0,C 180,E1 -14649.424,E2 -14649.424} C_VEL
LIN {X 0,Y 340.981,Z 320.788,A -85,B 0,C 180,E1 -14650.119,E2 -14650.119} C_VEL
LIN {X 0,Y 339.904,Z 332.139,A -85,B 0,C 180,E1 -14650.996,E2 -14650.996} C_VEL
LIN {X 0,Y 338.579,Z 343.806,A -85,B 0,C 180,E1 -14652.172,E2 -14652.172} C_VEL
LIN {X 0,Y 337.333,Z 354.757,A -85,B 0,C 180,E1 -14653.579,E2 -14653.579} C_VEL
LIN {X 0,Y 336.093,Z 364.538,A -85,B 0,C 180,E1 -14655.159,E2 -14655.159} C_VEL
LIN {X 0,Y 334.779,Z 373.474,A -85,B 0,C 180,E1 -14656.958,E2 -14656.958} C_VEL
LIN {X 0,Y 333.811,Z 380.669,A -85,B 0,C 180,E1 -14658.771,E2 -14658.771} C_VEL
LIN {X 0,Y 333.168,Z 385.522,A -85,B 0,C 180,E1 -14660.285,E2 -14660.285} C_VEL
LIN {X 0,Y 332.621,Z 390.239,A -85,B 0,C 180,E1 -14662.107,E2 -14662.107} C_VEL
LIN {X 0,Y 332.269,Z 393.85,A -85,B 0,C 180,E1 -14663.93,E2 -14663.93} C_VEL
LIN {X 0,Y 332.162,Z 395.715,A -85,B 0,C 180,E1 -14665.146,E2 -14665.146} C_VEL
LIN {X 0,Y 332.045,Z 397.12,A -85,B 0,C 180,E1 -14666.36,E2 -14666.36} C_VEL
LIN {X 0,Y 331.878,Z 398.734,A -85,B 0,C 180,E1 -14668.787,E2 -14668.787} C_VEL
LIN {X 0,Y 331.886,Z 398.967,A -85,B 0,C 180,E1 -14670.001,E2 -14670.001} C_VEL
LIN {X 0,Y 331.878,Z 398.776,A -85,B 0,C 180,E1 -14671.214,E2 -14671.214} C_VEL
LIN {X 0,Y 332.039,Z 397.215,A -85,B 0,C 180,E1 -14673.641,E2 -14673.641} C_VEL
LIN {X 0,Y 332.144,Z 395.852,A -85,B 0,C 180,E1 -14674.856,E2 -14674.856} C_VEL
LIN {X 0,Y 332.313,Z 393.663,A -85,B 0,C 180,E1 -14676.283,E2 -14676.283} C_VEL
LIN {X 0,Y 332.777,Z 389.068,A -85,B 0,C 180,E1 -14678.502,E2 -14678.502} C_VEL
LIN {X 0,Y 333.38,Z 384.033,A -85,B 0,C 180,E1 -14680.323,E2 -14680.323} C_VEL
LIN {X 0,Y 334.208,Z 377.695,A -85,B 0,C 180,E1 -14682.139,E2 -14682.139} C_VEL
LIN {X 0,Y 335.359,Z 369.764,A -85,B 0,C 180,E1 -14683.946,E2 -14683.946} C_VEL
LIN {X 0,Y 336.791,Z 359.9,A -85,B 0,C 180,E1 -14685.74,E2 -14685.74} C_VEL
LIN {X 0,Y 337.762,Z 350.723,A -85,B 0,C 180,E1 -14687.092,E2 -14687.092} C_VEL
LIN {X 0,Y 339.114,Z 339.302,A -85,B 0,C 180,E1 -14688.424,E2 -14688.424} C_VEL
LIN {X 0,Y 340.333,Z 328.089,A -85,B 0,C 180,E1 -14689.45,E2 -14689.45} C_VEL
LIN {X 0,Y 341.405,Z 315.454,A -85,B 0,C 180,E1 -14690.327,E2 -14690.327} C_VEL
LIN {X 0,Y 342.239,Z 302.789,A -85,B 0,C 180,E1 -14690.943,E2 -14690.943} C_VEL
LIN {X 0,Y 342.727,Z 289.767,A -85,B 0,C 180,E1 -14691.345,E2 -14691.345} C_VEL
LIN {X 0,Y 344.033,Z 219.033,A -85,B 0,C 180,E1 -14692.823,E2 -14692.823} C_VEL
LIN {X 0,Y 339.079,Z 193.604,A -85,B 0,C 180,E1 -14693.752,E2 -14693.752} C_VEL
LIN {X 0,Y 338.699,Z 192.657,A -85,B 0,C 180,E1 -14693.802,E2 -14693.802} C_VEL
LIN {X 0,Y 337.321,Z 189.659,A -85,B 0,C 180,E1 -14694.061,E2 -14694.061} C_VEL
LIN {X 0,Y 335.228,Z 186.839,A -85,B 0,C 180,E1 -14694.577,E2 -14694.577} C_VEL
LIN {X 0,Y 332.299,Z 183.964,A -85,B 0,C 180,E1 -14695.484,E2 -14695.484} C_VEL
LIN {X 0,Y 329.294,Z 180.552,A -85,B 0,C 180,E1 -14696.747,E2 -14696.747} C_VEL
LIN {X 0,Y 327.528,Z 176.73,A -85,B 0,C 180,E1 -14698.052,E2 -14698.052} C_VEL
LIN {X 0,Y 326.707,Z 172.808,A -85,B 0,C 180,E1 -14699.433,E2 -14699.433} C_VEL
LIN {X 0,Y 326.608,Z 172.791,A -85,B 0,C 180,E1 -14704.019,E2 -14704.019} C_VEL
LIN {X 0,Y 326.627,Z 172.799,A -85,B 0,C 180,E1 -14707.238,E2 -14707.238} C_VEL
LIN {X 0,Y 326.577,Z 172.787,A -85,B 0,C 180,E1 -14711.131,E2 -14711.131} C_VEL
LIN {X 0,Y 326.526,Z 172.803,A -85,B 0,C 180,E1 -14714.742,E2 -14714.742} C_VEL
LIN {X 0,Y 326.575,Z 172.785,A -85,B 0,C 180,E1 -14718.154,E2 -14718.154} C_VEL
LIN {X 0,Y 326.622,Z 172.799,A -85,B 0,C 180,E1 -14721.391,E2 -14721.391} C_VEL
LIN {X 0,Y 326.617,Z 172.756,A -85,B 0,C 180,E1 -14724.851,E2 -14724.851} C_VEL
LIN {X 0,Y 326.605,Z 172.788,A -85,B 0,C 180,E1 -14727.455,E2 -14727.455} C_VEL
LIN {X 0,Y 326.658,Z 172.793,A -85,B 0,C 180,E1 -14730.34,E2 -14730.34} C_VEL
LIN {X 0,Y 326.687,Z 172.791,A -85,B 0,C 180,E1 -14734.516,E2 -14734.516} C_VEL
LIN {X 0,Y 326.615,Z 172.789,A -85,B 0,C 180,E1 -14738.543,E2 -14738.543} C_VEL
LIN {X 0,Y 326.741,Z 172.784,A -85,B 0,C 180,E1 -14741.177,E2 -14741.177} C_VEL
LIN {X 0,Y 326.759,Z 172.77,A -85,B 0,C 180,E1 -14745.433,E2 -14745.433} C_VEL
LIN {X 0,Y 326.765,Z 172.777,A -85,B 0,C 180,E1 -14748.839,E2 -14748.839} C_VEL
LIN {X 0,Y 326.971,Z 172.749,A -85,B 0,C 180,E1 -14752.59,E2 -14752.59} C_VEL
LIN {X 0,Y 326.768,Z 172.78,A -85,B 0,C 180,E1 -14755.065,E2 -14755.065} C_VEL
LIN {X 0,Y 327.038,Z 172.731,A -85,B 0,C 180,E1 -14757.537,E2 -14757.537} C_VEL
LIN {X 0,Y 327.173,Z 172.73,A -85,B 0,C 180,E1 -14760,E2 -14760} C_VEL
LIN {X 0,Y 327.039,Z 172.743,A -85,B 0,C 180,E1 -14762.463,E2 -14762.463} C_VEL
LIN {X 0,Y 326.976,Z 172.75,A -85,B 0,C 180,E1 -14766.169,E2 -14766.169} C_VEL
LIN {X 0,Y 326.778,Z 172.771,A -85,B 0,C 180,E1 -14769.907,E2 -14769.907} C_VEL
LIN {X 0,Y 326.752,Z 172.783,A -85,B 0,C 180,E1 -14773.686,E2 -14773.686} C_VEL
LIN {X 0,Y 326.659,Z 172.781,A -85,B 0,C 180,E1 -14777.53,E2 -14777.53} C_VEL
LIN {X 0,Y 326.645,Z 172.794,A -85,B 0,C 180,E1 -14780.136,E2 -14780.136} C_VEL
LIN {X 0,Y 326.645,Z 172.784,A -85,B 0,C 180,E1 -14784.129,E2 -14784.129} C_VEL
LIN {X 0,Y 326.679,Z 172.794,A -85,B 0,C 180,E1 -14786.858,E2 -14786.858} C_VEL
LIN {X 0,Y 326.631,Z 172.793,A -85,B 0,C 180,E1 -14790.61,E2 -14790.61} C_VEL
LIN {X 0,Y 326.604,Z 172.792,A -85,B 0,C 180,E1 -14794.02,E2 -14794.02} C_VEL
LIN {X 0,Y 326.624,Z 172.763,A -85,B 0,C 180,E1 -14797.239,E2 -14797.239} C_VEL
LIN {X 0,Y 326.575,Z 172.805,A -85,B 0,C 180,E1 -14801.132,E2 -14801.132} C_VEL
LIN {X 0,Y 326.525,Z 172.811,A -85,B 0,C 180,E1 -14804.743,E2 -14804.743} C_VEL
LIN {X 0,Y 326.572,Z 172.804,A -85,B 0,C 180,E1 -14808.154,E2 -14808.154} C_VEL
LIN {X 0,Y 326.585,Z 172.781,A -85,B 0,C 180,E1 -14811.386,E2 -14811.386} C_VEL
LIN {X 0,Y 326.619,Z 172.795,A -85,B 0,C 180,E1 -14814.852,E2 -14814.852} C_VEL
LIN {X 0,Y 326.608,Z 172.798,A -85,B 0,C 180,E1 -14817.456,E2 -14817.456} C_VEL
LIN {X 0,Y 326.657,Z 172.979,A -85,B 0,C 180,E1 -14819.286,E2 -14819.286} C_VEL
LIN {X 0,Y 328.98,Z 183.593,A -85,B 0,C 180,E1 -14822.658,E2 -14822.658} C_VEL
LIN {X 0,Y 330.743,Z 193.069,A -85,B 0,C 180,E1 -14825.454,E2 -14825.454} C_VEL
LIN {X 0,Y 331.817,Z 197.59,A -85,B 0,C 180,E1 -14825.703,E2 -14825.703} C_VEL
LIN {X 0,Y 336.723,Z 224.298,A -85,B 0,C 180,E1 -14826.687,E2 -14826.687} C_VEL
LIN {X 0,Y 337.417,Z 229.784,A -85,B 0,C 180,E1 -14826.862,E2 -14826.862} C_VEL
LIN {X 0,Y 335.899,Z 301.103,A -85,B 0,C 180,E1 -14828.401,E2 -14828.401} C_VEL
LIN {X 0,Y 335.104,Z 314.277,A -85,B 0,C 180,E1 -14828.911,E2 -14828.911} C_VEL
LIN {X 0,Y 334.094,Z 326.381,A -85,B 0,C 180,E1 -14829.61,E2 -14829.61} C_VEL
LIN {X 0,Y 332.935,Z 338.598,A -85,B 0,C 180,E1 -14830.581,E2 -14830.581} C_VEL
LIN {X 0,Y 331.55,Z 350.158,A -85,B 0,C 180,E1 -14831.78,E2 -14831.78} C_VEL
LIN {X 0,Y 330.28,Z 359.928,A -85,B 0,C 180,E1 -14833.052,E2 -14833.052} C_VEL
LIN {X 0,Y 329.109,Z 369.073,A -85,B 0,C 180,E1 -14834.518,E2 -14834.518} C_VEL
LIN {X 0,Y 328.004,Z 376.92,A -85,B 0,C 180,E1 -14836.051,E2 -14836.051} C_VEL
LIN {X 0,Y 326.823,Z 384.581,A -85,B 0,C 180,E1 -14837.897,E2 -14837.897} C_VEL
LIN {X 0,Y 325.891,Z 391.646,A -85,B 0,C 180,E1 -14840.065,E2 -14840.065} C_VEL
LIN {X 0,Y 325.365,Z 396.344,A -85,B 0,C 180,E1 -14841.929,E2 -14841.929} C_VEL
LIN {X 0,Y 325.034,Z 400.381,A -85,B 0,C 180,E1 -14844.06,E2 -14844.06} C_VEL
LIN {X 0,Y 324.883,Z 403.17,A -85,B 0,C 180,E1 -14846.279,E2 -14846.279} C_VEL
LIN {X 0,Y 324.777,Z 404.762,A -85,B 0,C 180,E1 -14848.76,E2 -14848.76} C_VEL
LIN {X 0,Y 324.792,Z 404.975,A -85,B 0,C 180,E1 -14849.999,E2 -14849.999} C_VEL
LIN {X 0,Y 324.777,Z 404.756,A -85,B 0,C 180,E1 -14851.239,E2 -14851.239} C_VEL
LIN {X 0,Y 324.883,Z 403.157,A -85,B 0,C 180,E1 -14853.72,E2 -14853.72} C_VEL
LIN {X 0,Y 325.063,Z 400.276,A -85,B 0,C 180,E1 -14855.988,E2 -14855.988} C_VEL
LIN {X 0,Y 325.398,Z 396.302,A -85,B 0,C 180,E1 -14858.07,E2 -14858.07} C_VEL
LIN {X 0,Y 325.889,Z 391.593,A -85,B 0,C 180,E1 -14859.934,E2 -14859.934} C_VEL
LIN {X 0,Y 326.7,Z 385.635,A -85,B 0,C 180,E1 -14861.791,E2 -14861.791} C_VEL
LIN {X 0,Y 327.768,Z 378.212,A -85,B 0,C 180,E1 -14863.642,E2 -14863.642} C_VEL
LIN {X 0,Y 328.906,Z 370.647,A -85,B 0,C 180,E1 -14865.173,E2 -14865.173} C_VEL
LIN {X 0,Y 330.139,Z 360.982,A -85,B 0,C 180,E1 -14866.778,E2 -14866.778} C_VEL
LIN {X 0,Y 331.53,Z 350.002,A -85,B 0,C 180,E1 -14868.22,E2 -14868.22} C_VEL
LIN {X 0,Y 332.89,Z 338.406,A -85,B 0,C 180,E1 -14869.42,E2 -14869.42} C_VEL
LIN {X 0,Y 334.18,Z 326.097,A -85,B 0,C 180,E1 -14870.383,E2 -14870.383} C_VEL
LIN {X 0,Y 335.182,Z 313.13,A -85,B 0,C 180,E1 -14871.123,E2 -14871.123} C_VEL
LIN {X 0,Y 335.877,Z 300.527,A -85,B 0,C 180,E1 -14871.6,E2 -14871.6} C_VEL
LIN {X 0,Y 337.356,Z 228.177,A -85,B 0,C 180,E1 -14873.157,E2 -14873.157} C_VEL
LIN {X 0,Y 332.411,Z 200.717,A -85,B 0,C 180,E1 -14874.156,E2 -14874.156} C_VEL
LIN {X 0,Y 330.783,Z 193.269,A -85,B 0,C 180,E1 -14874.494,E2 -14874.494} C_VEL
LIN {X 0,Y 329.547,Z 186.613,A -85,B 0,C 180,E1 -14876.401,E2 -14876.401} C_VEL
LIN {X 0,Y 327.394,Z 176.337,A -85,B 0,C 180,E1 -14879.585,E2 -14879.585} C_VEL
LIN {X 0,Y 326.583,Z 172.837,A -85,B 0,C 180,E1 -14880.79,E2 -14880.79} C_VEL
LIN {X 0,Y 326.603,Z 172.788,A -85,B 0,C 180,E1 -14884.018,E2 -14884.018} C_VEL
LIN {X 0,Y 326.619,Z 172.785,A -85,B 0,C 180,E1 -14887.236,E2 -14887.236} C_VEL
LIN {X 0,Y 326.57,Z 172.808,A -85,B 0,C 180,E1 -14891.13,E2 -14891.13} C_VEL
LIN {X 0,Y 326.521,Z 172.813,A -85,B 0,C 180,E1 -14894.742,E2 -14894.742} C_VEL
LIN {X 0,Y 326.57,Z 172.803,A -85,B 0,C 180,E1 -14898.153,E2 -14898.153} C_VEL
LIN {X 0,Y 326.616,Z 172.783,A -85,B 0,C 180,E1 -14901.39,E2 -14901.39} C_VEL
LIN {X 0,Y 326.611,Z 172.774,A -85,B 0,C 180,E1 -14904.85,E2 -14904.85} C_VEL
LIN {X 0,Y 326.6,Z 172.803,A -85,B 0,C 180,E1 -14907.455,E2 -14907.455} C_VEL
LIN {X 0,Y 326.639,Z 172.787,A -85,B 0,C 180,E1 -14910.339,E2 -14910.339} C_VEL
LIN {X 0,Y 326.681,Z 172.789,A -85,B 0,C 180,E1 -14914.515,E2 -14914.515} C_VEL
LIN {X 0,Y 326.609,Z 172.801,A -85,B 0,C 180,E1 -14918.543,E2 -14918.543} C_VEL
LIN {X 0,Y 326.698,Z 172.777,A -85,B 0,C 180,E1 -14921.175,E2 -14921.175} C_VEL
LIN {X 0,Y 326.753,Z 172.782,A -85,B 0,C 180,E1 -14925.433,E2 -14925.433} C_VEL
LIN {X 0,Y 326.762,Z 172.767,A -85,B 0,C 180,E1 -14928.839,E2 -14928.839} C_VEL
LIN {X 0,Y 326.955,Z 172.758,A -85,B 0,C 180,E1 -14932.59,E2 -14932.59} C_VEL
LIN {X 0,Y 326.762,Z 172.764,A -85,B 0,C 180,E1 -14935.065,E2 -14935.065} C_VEL
LIN {X 0,Y 327.034,Z 172.744,A -85,B 0,C 180,E1 -14937.537,E2 -14937.537} C_VEL
LIN {X 0,Y 327.187,Z 172.728,A -85,B 0,C 180,E1 -14940,E2 -14940} C_VEL
LIN {X 0,Y 327.033,Z 172.732,A -85,B 0,C 180,E1 -14942.463,E2 -14942.463} C_VEL
LIN {X 0,Y 326.956,Z 172.752,A -85,B 0,C 180,E1 -14946.724,E2 -14946.724} C_VEL
LIN {X 0,Y 326.803,Z 172.759,A -85,B 0,C 180,E1 -14949.907,E2 -14949.907} C_VEL
LIN {X 0,Y 326.749,Z 172.78,A -85,B 0,C 180,E1 -14953.686,E2 -14953.686} C_VEL
LIN {X 0,Y 326.689,Z 172.785,A -85,B 0,C 180,E1 -14957.529,E2 -14957.529} C_VEL
LIN {X 0,Y 326.654,Z 172.793,A -85,B 0,C 180,E1 -14960.136,E2 -14960.136} C_VEL
LIN {X 0,Y 326.643,Z 172.795,A -85,B 0,C 180,E1 -14964.13,E2 -14964.13} C_VEL
LIN {X 0,Y 326.675,Z 172.784,A -85,B 0,C 180,E1 -14966.859,E2 -14966.859} C_VEL
LIN {X 0,Y 326.631,Z 172.798,A -85,B 0,C 180,E1 -14970.612,E2 -14970.612} C_VEL
LIN {X 0,Y 326.599,Z 172.768,A -85,B 0,C 180,E1 -14974.021,E2 -14974.021} C_VEL
LIN {X 0,Y 326.62,Z 172.782,A -85,B 0,C 180,E1 -14977.24,E2 -14977.24} C_VEL
LIN {X 0,Y 326.572,Z 172.801,A -85,B 0,C 180,E1 -14981.133,E2 -14981.133} C_VEL
LIN {X 0,Y 326.521,Z 172.793,A -85,B 0,C 180,E1 -14984.744,E2 -14984.744} C_VEL
LIN {X 0,Y 326.571,Z 172.798,A -85,B 0,C 180,E1 -14988.155,E2 -14988.155} C_VEL
LIN {X 0,Y 326.594,Z 172.789,A -85,B 0,C 180,E1 -14991.389,E2 -14991.389} C_VEL
LIN {X 0,Y 326.616,Z 172.785,A -85,B 0,C 180,E1 -14994.853,E2 -14994.853} C_VEL
LIN {X 0,Y 326.605,Z 172.802,A -85,B 0,C 180,E1 -14997.457,E2 -14997.457} C_VEL
LIN {X 0,Y 326.711,Z 172.927,A -85,B 0,C 180,E1 -15000.79,E2 -15000.79} C_VEL
LIN {X 0,Y 328.871,Z 183.161,A -85,B 0,C 180,E1 -15004.1,E2 -15004.1} C_VEL
LIN {X 0,Y 329.785,Z 187.777,A -85,B 0,C 180,E1 -15005.461,E2 -15005.461} C_VEL
LIN {X 0,Y 332.52,Z 195.056,A -85,B 0,C 180,E1 -15005.895,E2 -15005.895} C_VEL
LIN {X 0,Y 335.933,Z 211.506,A -85,B 0,C 180,E1 -15006.533,E2 -15006.533} C_VEL
LIN {X 0,Y 337.48,Z 220.84,A -85,B 0,C 180,E1 -15006.859,E2 -15006.859} C_VEL
LIN {X 0,Y 335.962,Z 295.828,A -85,B 0,C 180,E1 -15008.487,E2 -15008.487} C_VEL
LIN {X 0,Y 335.18,Z 308.841,A -85,B 0,C 180,E1 -15008.998,E2 -15008.998} C_VEL
LIN {X 0,Y 334.316,Z 320.861,A -85,B 0,C 180,E1 -15009.706,E2 -15009.706} C_VEL
LIN {X 0,Y 333.214,Z 332.21,A -85,B 0,C 180,E1 -15010.599,E2 -15010.599} C_VEL
LIN {X 0,Y 331.828,Z 343.876,A -85,B 0,C 180,E1 -15011.797,E2 -15011.797} C_VEL
LIN {X 0,Y 330.514,Z 354.826,A -85,B 0,C 180,E1 -15013.231,E2 -15013.231} C_VEL
LIN {X 0,Y 329.239,Z 364.606,A -85,B 0,C 180,E1 -15014.842,E2 -15014.842} C_VEL
LIN {X 0,Y 327.837,Z 373.542,A -85,B 0,C 180,E1 -15016.677,E2 -15016.677} C_VEL
LIN {X 0,Y 326.825,Z 380.736,A -85,B 0,C 180,E1 -15018.528,E2 -15018.528} C_VEL
LIN {X 0,Y 326.158,Z 385.589,A -85,B 0,C 180,E1 -15020.074,E2 -15020.074} C_VEL
LIN {X 0,Y 325.584,Z 390.305,A -85,B 0,C 180,E1 -15021.935,E2 -15021.935} C_VEL
LIN {X 0,Y 325.193,Z 393.916,A -85,B 0,C 180,E1 -15023.797,E2 -15023.797} C_VEL
LIN {X 0,Y 325.07,Z 395.781,A -85,B 0,C 180,E1 -15025.04,E2 -15025.04} C_VEL
LIN {X 0,Y 324.977,Z 397.185,A -85,B 0,C 180,E1 -15026.281,E2 -15026.281} C_VEL
LIN {X 0,Y 324.79,Z 398.799,A -85,B 0,C 180,E1 -15028.761,E2 -15028.761} C_VEL
LIN {X 0,Y 324.794,Z 399.032,A -85,B 0,C 180,E1 -15030.001,E2 -15030.001} C_VEL
LIN {X 0,Y 324.79,Z 398.84,A -85,B 0,C 180,E1 -15031.24,E2 -15031.24} C_VEL
LIN {X 0,Y 324.972,Z 397.279,A -85,B 0,C 180,E1 -15033.72,E2 -15033.72} C_VEL
LIN {X 0,Y 325.053,Z 395.916,A -85,B 0,C 180,E1 -15034.962,E2 -15034.962} C_VEL
LIN {X 0,Y 325.305,Z 393.142,A -85,B 0,C 180,E1 -15036.762,E2 -15036.762} C_VEL
LIN {X 0,Y 325.743,Z 389.132,A -85,B 0,C 180,E1 -15038.687,E2 -15038.687} C_VEL
LIN {X 0,Y 326.365,Z 384.096,A -85,B 0,C 180,E1 -15040.547,E2 -15040.547} C_VEL
LIN {X 0,Y 327.233,Z 377.758,A -85,B 0,C 180,E1 -15042.402,E2 -15042.402} C_VEL
LIN {X 0,Y 328.467,Z 369.826,A -85,B 0,C 180,E1 -15044.245,E2 -15044.245} C_VEL
LIN {X 0,Y 329.933,Z 359.962,A -85,B 0,C 180,E1 -15046.076,E2 -15046.076} C_VEL
LIN {X 0,Y 330.982,Z 350.784,A -85,B 0,C 180,E1 -15047.453,E2 -15047.453} C_VEL
LIN {X 0,Y 332.402,Z 339.362,A -85,B 0,C 180,E1 -15048.81,E2 -15048.81} C_VEL
LIN {X 0,Y 333.66,Z 328.147,A -85,B 0,C 180,E1 -15049.855,E2 -15049.855} C_VEL
LIN {X 0,Y 334.771,Z 315.51,A -85,B 0,C 180,E1 -15050.748,E2 -15050.748} C_VEL
LIN {X 0,Y 335.631,Z 302.841,A -85,B 0,C 180,E1 -15051.376,E2 -15051.376} C_VEL
LIN {X 0,Y 336.123,Z 289.812,A -85,B 0,C 180,E1 -15051.786,E2 -15051.786} C_VEL
LIN {X 0,Y 337.486,Z 219.861,A -85,B 0,C 180,E1 -15053.274,E2 -15053.274} C_VEL
LIN {X 0,Y 332.907,Z 196.197,A -85,B 0,C 180,E1 -15054.161,E2 -15054.161} C_VEL
LIN {X 0,Y 329.824,Z 187.955,A -85,B 0,C 180,E1 -15054.63,E2 -15054.63} C_VEL
LIN {X 0,Y 329.084,Z 184.181,A -85,B 0,C 180,E1 -15055.697,E2 -15055.697} C_VEL
LIN {X 0,Y 327.528,Z 176.73,A -85,B 0,C 180,E1 -15058.052,E2 -15058.052} C_VEL
LIN {X 0,Y 326.468,Z 175.195,A -85,B 0,C 180,E1 -15058.671,E2 -15058.671} C_VEL
LIN {X 0,Y 324.632,Z 174.282,A -85,B 0,C 180,E1 -15059.287,E2 -15059.287} C_VEL
LIN {X 0,Y 320.721,Z 173.68,A -85,B 0,C 180,E1 -15060.563,E2 -15060.563} C_VEL
LIN {X 0,Y 319.631,Z 173.668,A -85,B 0,C 180,E1 -15061.261,E2 -15061.261} C_VEL
LIN {X 0,Y 319.538,Z 173.671,A -85,B 0,C 180,E1 -15061.503,E2 -15061.503} C_VEL
LIN {X 0,Y 319.56,Z 173.663,A -85,B 0,C 180,E1 -15064.876,E2 -15064.876} C_VEL
LIN {X 0,Y 319.557,Z 173.675,A -85,B 0,C 180,E1 -15068.01,E2 -15068.01} C_VEL
LIN {X 0,Y 319.525,Z 173.672,A -85,B 0,C 180,E1 -15071.596,E2 -15071.596} C_VEL
LIN {X 0,Y 319.487,Z 173.671,A -85,B 0,C 180,E1 -15075.257,E2 -15075.257} C_VEL
LIN {X 0,Y 319.527,Z 173.672,A -85,B 0,C 180,E1 -15078.711,E2 -15078.711} C_VEL
LIN {X 0,Y 319.56,Z 173.667,A -85,B 0,C 180,E1 -15082.347,E2 -15082.347} C_VEL
LIN {X 0,Y 319.557,Z 173.634,A -85,B 0,C 180,E1 -15085.123,E2 -15085.123} C_VEL
LIN {X 0,Y 319.568,Z 173.676,A -85,B 0,C 180,E1 -15089.058,E2 -15089.058} C_VEL
LIN {X 0,Y 319.605,Z 173.662,A -85,B 0,C 180,E1 -15092.498,E2 -15092.498} C_VEL
LIN {X 0,Y 319.6,Z 173.674,A -85,B 0,C 180,E1 -15095.303,E2 -15095.303} C_VEL
LIN {X 0,Y 319.598,Z 173.666,A -85,B 0,C 180,E1 -15099.4,E2 -15099.4} C_VEL
LIN {X 0,Y 319.654,Z 173.664,A -85,B 0,C 180,E1 -15102.073,E2 -15102.073} C_VEL
LIN {X 0,Y 319.728,Z 173.653,A -85,B 0,C 180,E1 -15106.007,E2 -15106.007} C_VEL
LIN {X 0,Y 319.753,Z 173.64,A -85,B 0,C 180,E1 -15109.873,E2 -15109.873} C_VEL
LIN {X 0,Y 319.928,Z 173.627,A -85,B 0,C 180,E1 -15112.426,E2 -15112.426} C_VEL
LIN {X 0,Y 319.738,Z 173.655,A -85,B 0,C 180,E1 -15114.956,E2 -15114.956} C_VEL
LIN {X 0,Y 319.982,Z 173.61,A -85,B 0,C 180,E1 -15117.482,E2 -15117.482} C_VEL
LIN {X 0,Y 320.126,Z 173.608,A -85,B 0,C 180,E1 -15120,E2 -15120} C_VEL
LIN {X 0,Y 319.982,Z 173.622,A -85,B 0,C 180,E1 -15122.518,E2 -15122.518} C_VEL
LIN {X 0,Y 319.93,Z 173.627,A -85,B 0,C 180,E1 -15126.306,E2 -15126.306} C_VEL
LIN {X 0,Y 319.731,Z 173.648,A -85,B 0,C 180,E1 -15130.128,E2 -15130.128} C_VEL
LIN {X 0,Y 319.726,Z 173.657,A -85,B 0,C 180,E1 -15133.992,E2 -15133.992} C_VEL
LIN {X 0,Y 319.62,Z 173.656,A -85,B 0,C 180,E1 -15137.929,E2 -15137.929} C_VEL
LIN {X 0,Y 319.593,Z 173.674,A -85,B 0,C 180,E1 -15140.6,E2 -15140.6} C_VEL
LIN {X 0,Y 319.599,Z 173.663,A -85,B 0,C 180,E1 -15144.697,E2 -15144.697} C_VEL
LIN {X 0,Y 319.608,Z 173.669,A -85,B 0,C 180,E1 -15148.41,E2 -15148.41} C_VEL
LIN {X 0,Y 319.528,Z 173.683,A -85,B 0,C 180,E1 -15151.862,E2 -15151.862} C_VEL
LIN {X 0,Y 319.577,Z 173.644,A -85,B 0,C 180,E1 -15155.543,E2 -15155.543} C_VEL
LIN {X 0,Y 319.554,Z 173.653,A -85,B 0,C 180,E1 -15158.011,E2 -15158.011} C_VEL
LIN {X 0,Y 319.523,Z 173.68,A -85,B 0,C 180,E1 -15161.597,E2 -15161.597} C_VEL
LIN {X 0,Y 319.486,Z 173.689,A -85,B 0,C 180,E1 -15165.257,E2 -15165.257} C_VEL
LIN {X 0,Y 319.524,Z 173.686,A -85,B 0,C 180,E1 -15168.712,E2 -15168.712} C_VEL
LIN {X 0,Y 319.546,Z 173.661,A -85,B 0,C 180,E1 -15172.352,E2 -15172.352} C_VEL
LIN {X 0,Y 319.56,Z 173.671,A -85,B 0,C 180,E1 -15175.124,E2 -15175.124} C_VEL
LIN {X 0,Y 319.574,Z 173.788,A -85,B 0,C 180,E1 -15178.786,E2 -15178.786} C_VEL
LIN {X 0,Y 321.747,Z 183.523,A -85,B 0,C 180,E1 -15181.99,E2 -15181.99} C_VEL
LIN {X 0,Y 323.643,Z 193.14,A -85,B 0,C 180,E1 -15184.897,E2 -15184.897} C_VEL
LIN {X 0,Y 325.191,Z 198.178,A -85,B 0,C 180,E1 -15185.19,E2 -15185.19} C_VEL
LIN {X 0,Y 330.076,Z 224.38,A -85,B 0,C 180,E1 -15186.192,E2 -15186.192} C_VEL
LIN {X 0,Y 330.892,Z 230.769,A -85,B 0,C 180,E1 -15186.402,E2 -15186.402} C_VEL
LIN {X 0,Y 329.306,Z 301.051,A -85,B 0,C 180,E1 -15187.946,E2 -15187.946} C_VEL
LIN {X 0,Y 328.504,Z 314.221,A -85,B 0,C 180,E1 -15188.467,E2 -15188.467} C_VEL
LIN {X 0,Y 327.451,Z 326.323,A -85,B 0,C 180,E1 -15189.177,E2 -15189.177} C_VEL
LIN {X 0,Y 326.254,Z 338.537,A -85,B 0,C 180,E1 -15190.167,E2 -15190.167} C_VEL
LIN {X 0,Y 324.795,Z 350.096,A -85,B 0,C 180,E1 -15191.387,E2 -15191.387} C_VEL
LIN {X 0,Y 323.419,Z 360.345,A -85,B 0,C 180,E1 -15192.754,E2 -15192.754} C_VEL
LIN {X 0,Y 322.227,Z 369.01,A -85,B 0,C 180,E1 -15194.179,E2 -15194.179} C_VEL
LIN {X 0,Y 321.088,Z 376.857,A -85,B 0,C 180,E1 -15195.745,E2 -15195.745} C_VEL
LIN {X 0,Y 319.856,Z 384.518,A -85,B 0,C 180,E1 -15197.629,E2 -15197.629} C_VEL
LIN {X 0,Y 319.15,Z 389.768,A -85,B 0,C 180,E1 -15199.212,E2 -15199.212} C_VEL
LIN {X 0,Y 318.493,Z 394.854,A -85,B 0,C 180,E1 -15201.114,E2 -15201.114} C_VEL
LIN {X 0,Y 318.073,Z 398.802,A -85,B 0,C 180,E1 -15203.019,E2 -15203.019} C_VEL
LIN {X 0,Y 317.861,Z 401.718,A -85,B 0,C 180,E1 -15204.926,E2 -15204.926} C_VEL
LIN {X 0,Y 317.796,Z 403.105,A -85,B 0,C 180,E1 -15206.195,E2 -15206.195} C_VEL
LIN {X 0,Y 317.734,Z 404.095,A -85,B 0,C 180,E1 -15207.464,E2 -15207.464} C_VEL
LIN {X 0,Y 317.691,Z 404.698,A -85,B 0,C 180,E1 -15208.732,E2 -15208.732} C_VEL
LIN {X 0,Y 317.704,Z 404.91,A -85,B 0,C 180,E1 -15209.999,E2 -15209.999} C_VEL
LIN {X 0,Y 317.691,Z 404.691,A -85,B 0,C 180,E1 -15211.267,E2 -15211.267} C_VEL
LIN {X 0,Y 317.733,Z 404.084,A -85,B 0,C 180,E1 -15212.535,E2 -15212.535} C_VEL
LIN {X 0,Y 317.796,Z 403.091,A -85,B 0,C 180,E1 -15213.803,E2 -15213.803} C_VEL
LIN {X 0,Y 317.981,Z 400.452,A -85,B 0,C 180,E1 -15215.962,E2 -15215.962} C_VEL
LIN {X 0,Y 318.332,Z 396.236,A -85,B 0,C 180,E1 -15218.25,E2 -15218.25} C_VEL
LIN {X 0,Y 318.888,Z 391.526,A -85,B 0,C 180,E1 -15220.154,E2 -15220.154} C_VEL
LIN {X 0,Y 319.719,Z 385.568,A -85,B 0,C 180,E1 -15222.053,E2 -15222.053} C_VEL
LIN {X 0,Y 320.851,Z 378.145,A -85,B 0,C 180,E1 -15223.942,E2 -15223.942} C_VEL
LIN {X 0,Y 322.022,Z 370.579,A -85,B 0,C 180,E1 -15225.506,E2 -15225.506} C_VEL
LIN {X 0,Y 323.273,Z 361.29,A -85,B 0,C 180,E1 -15227.086,E2 -15227.086} C_VEL
LIN {X 0,Y 324.631,Z 351.226,A -85,B 0,C 180,E1 -15228.458,E2 -15228.458} C_VEL
LIN {X 0,Y 326.024,Z 339.92,A -85,B 0,C 180,E1 -15229.682,E2 -15229.682} C_VEL
LIN {X 0,Y 327.286,Z 328.185,A -85,B 0,C 180,E1 -15230.668,E2 -15230.668} C_VEL
LIN {X 0,Y 328.384,Z 315.342,A -85,B 0,C 180,E1 -15231.458,E2 -15231.458} C_VEL
LIN {X 0,Y 329.168,Z 302.738,A -85,B 0,C 180,E1 -15231.98,E2 -15231.98} C_VEL
LIN {X 0,Y 329.809,Z 280.139,A -85,B 0,C 180,E1 -15232.512,E2 -15232.512} C_VEL
LIN {X 0,Y 330.796,Z 229.007,A -85,B 0,C 180,E1 -15233.623,E2 -15233.623} C_VEL
LIN {X 0,Y 325.785,Z 201.133,A -85,B 0,C 180,E1 -15234.667,E2 -15234.667} C_VEL
LIN {X 0,Y 324.329,Z 195.317,A -85,B 0,C 180,E1 -15234.924,E2 -15234.924} C_VEL
LIN {X 0,Y 323.586,Z 192.984,A -85,B 0,C 180,E1 -15235.11,E2 -15235.11} C_VEL
LIN {X 0,Y 321.466,Z 182.241,A -85,B 0,C 180,E1 -15238.391,E2 -15238.391} C_VEL
LIN {X 0,Y 319.532,Z 173.731,A -85,B 0,C 180,E1 -15241.242,E2 -15241.242} C_VEL
LIN {X 0,Y 319.556,Z 173.672,A -85,B 0,C 180,E1 -15244.875,E2 -15244.875} C_VEL
LIN {X 0,Y 319.53,Z 173.66,A -85,B 0,C 180,E1 -15248.012,E2 -15248.012} C_VEL
LIN {X 0,Y 319.519,Z 173.683,A -85,B 0,C 180,E1 -15251.595,E2 -15251.595} C_VEL
LIN {X 0,Y 319.482,Z 173.688,A -85,B 0,C 180,E1 -15255.256,E2 -15255.256} C_VEL
LIN {X 0,Y 319.522,Z 173.683,A -85,B 0,C 180,E1 -15258.711,E2 -15258.711} C_VEL
LIN {X 0,Y 319.554,Z 173.646,A -85,B 0,C 180,E1 -15262.347,E2 -15262.347} C_VEL
LIN {X 0,Y 319.552,Z 173.656,A -85,B 0,C 180,E1 -15265.122,E2 -15265.122} C_VEL
LIN {X 0,Y 319.558,Z 173.675,A -85,B 0,C 180,E1 -15269.058,E2 -15269.058} C_VEL
LIN {X 0,Y 319.597,Z 173.673,A -85,B 0,C 180,E1 -15272.497,E2 -15272.497} C_VEL
LIN {X 0,Y 319.593,Z 173.663,A -85,B 0,C 180,E1 -15275.303,E2 -15275.303} C_VEL
LIN {X 0,Y 319.587,Z 173.674,A -85,B 0,C 180,E1 -15279.399,E2 -15279.399} C_VEL
LIN {X 0,Y 319.614,Z 173.657,A -85,B 0,C 180,E1 -15282.071,E2 -15282.071} C_VEL
LIN {X 0,Y 319.723,Z 173.657,A -85,B 0,C 180,E1 -15286.007,E2 -15286.007} C_VEL
LIN {X 0,Y 319.748,Z 173.646,A -85,B 0,C 180,E1 -15289.873,E2 -15289.873} C_VEL
LIN {X 0,Y 319.915,Z 173.637,A -85,B 0,C 180,E1 -15292.426,E2 -15292.426} C_VEL
LIN {X 0,Y 319.732,Z 173.64,A -85,B 0,C 180,E1 -15294.956,E2 -15294.956} C_VEL
LIN {X 0,Y 319.977,Z 173.623,A -85,B 0,C 180,E1 -15297.482,E2 -15297.482} C_VEL
LIN {X 0,Y 320.139,Z 173.606,A -85,B 0,C 180,E1 -15300,E2 -15300} C_VEL
LIN {X 0,Y 319.977,Z 173.61,A -85,B 0,C 180,E1 -15302.518,E2 -15302.518} C_VEL
LIN {X 0,Y 319.916,Z 173.631,A -85,B 0,C 180,E1 -15306.716,E2 -15306.716} C_VEL
LIN {X 0,Y 319.747,Z 173.639,A -85,B 0,C 180,E1 -15310.128,E2 -15310.128} C_VEL
LIN {X 0,Y 319.721,Z 173.646,A -85,B 0,C 180,E1 -15314.724,E2 -15314.724} C_VEL
LIN {X 0,Y 319.68,Z 173.663,A -85,B 0,C 180,E1 -15319.038,E2 -15319.038} C_VEL
LIN {X 0,Y 319.561,Z 173.672,A -85,B 0,C 180,E1 -15323.32,E2 -15323.32} C_VEL
LIN {X 0,Y 319.626,Z 173.668,A -85,B 0,C 180,E1 -15326.089,E2 -15326.089} C_VEL
LIN {X 0,Y 319.581,Z 173.672,A -85,B 0,C 180,E1 -15328.935,E2 -15328.935} C_VEL
LIN {X 0,Y 319.525,Z 173.678,A -85,B 0,C 180,E1 -15331.863,E2 -15331.863} C_VEL
LIN {X 0,Y 319.572,Z 173.634,A -85,B 0,C 180,E1 -15335.544,E2 -15335.544} C_VEL
LIN {X 0,Y 319.55,Z 173.67,A -85,B 0,C 180,E1 -15338.011,E2 -15338.011} C_VEL
LIN {X 0,Y 319.52,Z 173.67,A -85,B 0,C 180,E1 -15341.598,E2 -15341.598} C_VEL
LIN {X 0,Y 319.482,Z 173.678,A -85,B 0,C 180,E1 -15345.258,E2 -15345.258} C_VEL
LIN {X 0,Y 319.524,Z 173.67,A -85,B 0,C 180,E1 -15348.713,E2 -15348.713} C_VEL
LIN {X 0,Y 319.551,Z 173.679,A -85,B 0,C 180,E1 -15352.351,E2 -15352.351} C_VEL
LIN {X 0,Y 319.557,Z 173.663,A -85,B 0,C 180,E1 -15355.125,E2 -15355.125} C_VEL
LIN {X 0,Y 319.568,Z 173.668,A -85,B 0,C 180,E1 -15359.059,E2 -15359.059} C_VEL
LIN {X 0,Y 319.647,Z 173.836,A -85,B 0,C 180,E1 -15360.351,E2 -15360.351} C_VEL
LIN {X 0,Y 321.757,Z 183.548,A -85,B 0,C 180,E1 -15363.579,E2 -15363.579} C_VEL
LIN {X 0,Y 322.638,Z 187.97,A -85,B 0,C 180,E1 -15364.895,E2 -15364.895} C_VEL
LIN {X 0,Y 326.786,Z 199.063,A -85,B 0,C 180,E1 -15365.538,E2 -15365.538} C_VEL
LIN {X 0,Y 330.953,Z 221.215,A -85,B 0,C 180,E1 -15366.382,E2 -15366.382} C_VEL
LIN {X 0,Y 329.38,Z 295.908,A -85,B 0,C 180,E1 -15368.035,E2 -15368.035} C_VEL
LIN {X 0,Y 328.535,Z 309.678,A -85,B 0,C 180,E1 -15368.594,E2 -15368.594} C_VEL
LIN {X 0,Y 327.57,Z 322.03,A -85,B 0,C 180,E1 -15369.351,E2 -15369.351} C_VEL
LIN {X 0,Y 326.322,Z 333.867,A -85,B 0,C 180,E1 -15370.336,E2 -15370.336} C_VEL
LIN {X 0,Y 324.917,Z 345.235,A -85,B 0,C 180,E1 -15371.559,E2 -15371.559} C_VEL
LIN {X 0,Y 323.618,Z 355.599,A -85,B 0,C 180,E1 -15372.972,E2 -15372.972} C_VEL
LIN {X 0,Y 322.398,Z 364.674,A -85,B 0,C 180,E1 -15374.513,E2 -15374.513} C_VEL
LIN {X 0,Y 320.914,Z 373.61,A -85,B 0,C 180,E1 -15376.384,E2 -15376.384} C_VEL
LIN {X 0,Y 319.864,Z 380.803,A -85,B 0,C 180,E1 -15378.274,E2 -15378.274} C_VEL
LIN {X 0,Y 319.158,Z 385.655,A -85,B 0,C 180,E1 -15379.854,E2 -15379.854} C_VEL
LIN {X 0,Y 318.531,Z 390.371,A -85,B 0,C 180,E1 -15381.755,E2 -15381.755} C_VEL
LIN {X 0,Y 318.088,Z 394.314,A -85,B 0,C 180,E1 -15383.858,E2 -15383.858} C_VEL
LIN {X 0,Y 317.889,Z 397.25,A -85,B 0,C 180,E1 -15386.198,E2 -15386.198} C_VEL
LIN {X 0,Y 317.704,Z 398.864,A -85,B 0,C 180,E1 -15388.733,E2 -15388.733} C_VEL
LIN {X 0,Y 317.705,Z 399.097,A -85,B 0,C 180,E1 -15390.001,E2 -15390.001} C_VEL
LIN {X 0,Y 317.704,Z 398.905,A -85,B 0,C 180,E1 -15391.268,E2 -15391.268} C_VEL
LIN {X 0,Y 317.883,Z 397.344,A -85,B 0,C 180,E1 -15393.803,E2 -15393.803} C_VEL
LIN {X 0,Y 318.11,Z 394.43,A -85,B 0,C 180,E1 -15396.18,E2 -15396.18} C_VEL
LIN {X 0,Y 318.529,Z 390.616,A -85,B 0,C 180,E1 -15398.246,E2 -15398.246} C_VEL
LIN {X 0,Y 319.129,Z 385.965,A -85,B 0,C 180,E1 -15400.148,E2 -15400.148} C_VEL
LIN {X 0,Y 320.138,Z 378.956,A -85,B 0,C 180,E1 -15402.36,E2 -15402.36} C_VEL
LIN {X 0,Y 321.352,Z 371.361,A -85,B 0,C 180,E1 -15404.243,E2 -15404.243} C_VEL
LIN {X 0,Y 322.803,Z 361.804,A -85,B 0,C 180,E1 -15406.117,E2 -15406.117} C_VEL
LIN {X 0,Y 324.052,Z 351.942,A -85,B 0,C 180,E1 -15407.676,E2 -15407.676} C_VEL
LIN {X 0,Y 325.507,Z 340.847,A -85,B 0,C 180,E1 -15409.06,E2 -15409.06} C_VEL
LIN {X 0,Y 326.8,Z 329.97,A -85,B 0,C 180,E1 -15410.126,E2 -15410.126} C_VEL
LIN {X 0,Y 327.954,Z 317.955,A -85,B 0,C 180,E1 -15411.036,E2 -15411.036} C_VEL
LIN {X 0,Y 328.859,Z 305.622,A -85,B 0,C 180,E1 -15411.715,E2 -15411.715} C_VEL
LIN {X 0,Y 329.546,Z 292.864,A -85,B 0,C 180,E1 -15412.161,E2 -15412.161} C_VEL
LIN {X 0,Y 330.985,Z 221.025,A -85,B 0,C 180,E1 -15413.733,E2 -15413.733} C_VEL
LIN {X 0,Y 326.667,Z 198.577,A -85,B 0,C 180,E1 -15414.598,E2 -15414.598} C_VEL
LIN {X 0,Y 322.644,Z 187.984,A -85,B 0,C 180,E1 -15415.218,E2 -15415.218} C_VEL
LIN {X 0,Y 321.005,Z 179.932,A -85,B 0,C 180,E1 -15417.708,E2 -15417.708} C_VEL
LIN {X 0,Y 319.667,Z 173.743,A -85,B 0,C 180,E1 -15419.829,E2 -15419.829} C_VEL
LIN {X 0,Y 319.538,Z 173.671,A -85,B 0,C 180,E1 -15421.503,E2 -15421.503} C_VEL
LIN {X 0,Y 318.851,Z 173.768,A -85,B 0,C 180,E1 -15422.554,E2 -15422.554} C_VEL
LIN {X 0,Y 315.987,Z 174.11,A -85,B 0,C 180,E1 -15424.265,E2 -15424.265} C_VEL
LIN {X 0,Y 313.589,Z 174.409,A -85,B 0,C 180,E1 -15425.651,E2 -15425.651} C_VEL
LIN {X 0,Y 312.588,Z 174.547,A -85,B 0,C 180,E1 -15426.725,E2 -15426.725} C_VEL
LIN {X 0,Y 312.521,Z 174.552,A -85,B 0,C 180,E1 -15427.089,E2 -15427.089} C_VEL
LIN {X 0,Y 312.489,Z 174.536,A -85,B 0,C 180,E1 -15430.709,E2 -15430.709} C_VEL
LIN {X 0,Y 312.451,Z 174.56,A -85,B 0,C 180,E1 -15434.209,E2 -15434.209} C_VEL
LIN {X 0,Y 312.483,Z 174.537,A -85,B 0,C 180,E1 -15437.918,E2 -15437.918} C_VEL
LIN {X 0,Y 312.502,Z 174.557,A -85,B 0,C 180,E1 -15440.971,E2 -15440.971} C_VEL
LIN {X 0,Y 312.529,Z 174.512,A -85,B 0,C 180,E1 -15444.22,E2 -15444.22} C_VEL
LIN {X 0,Y 312.502,Z 174.543,A -85,B 0,C 180,E1 -15447.333,E2 -15447.333} C_VEL
LIN {X 0,Y 312.549,Z 174.548,A -85,B 0,C 180,E1 -15451.276,E2 -15451.276} C_VEL
LIN {X 0,Y 312.582,Z 174.547,A -85,B 0,C 180,E1 -15454.71,E2 -15454.71} C_VEL
LIN {X 0,Y 312.533,Z 174.544,A -85,B 0,C 180,E1 -15458.912,E2 -15458.912} C_VEL
LIN {X 0,Y 312.635,Z 174.543,A -85,B 0,C 180,E1 -15461.656,E2 -15461.656} C_VEL
LIN {X 0,Y 312.69,Z 174.525,A -85,B 0,C 180,E1 -15465.686,E2 -15465.686} C_VEL
LIN {X 0,Y 312.698,Z 174.52,A -85,B 0,C 180,E1 -15469.642,E2 -15469.642} C_VEL
LIN {X 0,Y 312.868,Z 174.504,A -85,B 0,C 180,E1 -15472.254,E2 -15472.254} C_VEL
LIN {X 0,Y 312.709,Z 174.53,A -85,B 0,C 180,E1 -15474.842,E2 -15474.842} C_VEL
LIN {X 0,Y 312.985,Z 174.486,A -85,B 0,C 180,E1 -15478.713,E2 -15478.713} C_VEL
LIN {X 0,Y 312.983,Z 174.5,A -85,B 0,C 180,E1 -15481.287,E2 -15481.287} C_VEL
LIN {X 0,Y 312.704,Z 174.515,A -85,B 0,C 180,E1 -15485.158,E2 -15485.158} C_VEL
LIN {X 0,Y 312.886,Z 174.504,A -85,B 0,C 180,E1 -15486.448,E2 -15486.448} C_VEL
LIN {X 0,Y 312.681,Z 174.525,A -85,B 0,C 180,E1 -15490.359,E2 -15490.359} C_VEL
LIN {X 0,Y 312.663,Z 174.538,A -85,B 0,C 180,E1 -15494.865,E2 -15494.865} C_VEL
LIN {X 0,Y 312.587,Z 174.539,A -85,B 0,C 180,E1 -15499.216,E2 -15499.216} C_VEL
LIN {X 0,Y 312.522,Z 174.549,A -85,B 0,C 180,E1 -15502.78,E2 -15502.78} C_VEL
LIN {X 0,Y 312.599,Z 174.545,A -85,B 0,C 180,E1 -15505.936,E2 -15505.936} C_VEL
LIN {X 0,Y 312.535,Z 174.544,A -85,B 0,C 180,E1 -15509.651,E2 -15509.651} C_VEL
LIN {X 0,Y 312.517,Z 174.548,A -85,B 0,C 180,E1 -15513.689,E2 -15513.689} C_VEL
LIN {X 0,Y 312.523,Z 174.519,A -85,B 0,C 180,E1 -15517.386,E2 -15517.386} C_VEL
LIN {X 0,Y 312.488,Z 174.561,A -85,B 0,C 180,E1 -15520.71,E2 -15520.71} C_VEL
LIN {X 0,Y 312.45,Z 174.561,A -85,B 0,C 180,E1 -15524.21,E2 -15524.21} C_VEL
LIN {X 0,Y 312.481,Z 174.559,A -85,B 0,C 180,E1 -15527.919,E2 -15527.919} C_VEL
LIN {X 0,Y 312.476,Z 174.539,A -85,B 0,C 180,E1 -15530.968,E2 -15530.968} C_VEL
LIN {X 0,Y 312.531,Z 174.558,A -85,B 0,C 180,E1 -15534.221,E2 -15534.221} C_VEL
LIN {X 0,Y 312.521,Z 174.597,A -85,B 0,C 180,E1 -15538.245,E2 -15538.245} C_VEL
LIN {X 0,Y 314.757,Z 184.711,A -85,B 0,C 180,E1 -15541.695,E2 -15541.695} C_VEL
LIN {X 0,Y 316.437,Z 193.062,A -85,B 0,C 180,E1 -15544.283,E2 -15544.283} C_VEL
LIN {X 0,Y 318.919,Z 200.13,A -85,B 0,C 180,E1 -15544.716,E2 -15544.716} C_VEL
LIN {X 0,Y 323.665,Z 225.808,A -85,B 0,C 180,E1 -15545.725,E2 -15545.725} C_VEL
LIN {X 0,Y 324.372,Z 231.281,A -85,B 0,C 180,E1 -15545.912,E2 -15545.912} C_VEL
LIN {X 0,Y 322.758,Z 301,A -85,B 0,C 180,E1 -15547.474,E2 -15547.474} C_VEL
LIN {X 0,Y 321.927,Z 314.165,A -85,B 0,C 180,E1 -15548.004,E2 -15548.004} C_VEL
LIN {X 0,Y 320.826,Z 326.265,A -85,B 0,C 180,E1 -15548.727,E2 -15548.727} C_VEL
LIN {X 0,Y 319.582,Z 338.477,A -85,B 0,C 180,E1 -15549.735,E2 -15549.735} C_VEL
LIN {X 0,Y 318.08,Z 350.035,A -85,B 0,C 180,E1 -15550.98,E2 -15550.98} C_VEL
LIN {X 0,Y 316.595,Z 360.444,A -85,B 0,C 180,E1 -15552.395,E2 -15552.395} C_VEL
LIN {X 0,Y 315.38,Z 368.948,A -85,B 0,C 180,E1 -15553.826,E2 -15553.826} C_VEL
LIN {X 0,Y 314.197,Z 376.794,A -85,B 0,C 180,E1 -15555.425,E2 -15555.425} C_VEL
LIN {X 0,Y 312.906,Z 384.454,A -85,B 0,C 180,E1 -15557.35,E2 -15557.35} C_VEL
LIN {X 0,Y 311.896,Z 391.519,A -85,B 0,C 180,E1 -15559.614,E2 -15559.614} C_VEL
LIN {X 0,Y 311.263,Z 396.216,A -85,B 0,C 180,E1 -15561.56,E2 -15561.56} C_VEL
LIN {X 0,Y 310.907,Z 399.804,A -85,B 0,C 180,E1 -15563.51,E2 -15563.51} C_VEL
LIN {X 0,Y 310.782,Z 401.654,A -85,B 0,C 180,E1 -15564.81,E2 -15564.81} C_VEL
LIN {X 0,Y 310.712,Z 403.04,A -85,B 0,C 180,E1 -15566.109,E2 -15566.109} C_VEL
LIN {X 0,Y 310.659,Z 404.03,A -85,B 0,C 180,E1 -15567.406,E2 -15567.406} C_VEL
LIN {X 0,Y 310.608,Z 404.633,A -85,B 0,C 180,E1 -15568.703,E2 -15568.703} C_VEL
LIN {X 0,Y 310.617,Z 404.845,A -85,B 0,C 180,E1 -15569.999,E2 -15569.999} C_VEL
LIN {X 0,Y 310.658,Z 404.019,A -85,B 0,C 180,E1 -15572.593,E2 -15572.593} C_VEL
LIN {X 0,Y 310.712,Z 403.026,A -85,B 0,C 180,E1 -15573.89,E2 -15573.89} C_VEL
LIN {X 0,Y 310.873,Z 400.674,A -85,B 0,C 180,E1 -15575.889,E2 -15575.889} C_VEL
LIN {X 0,Y 311.163,Z 397.481,A -85,B 0,C 180,E1 -15577.788,E2 -15577.788} C_VEL
LIN {X 0,Y 311.653,Z 393.153,A -85,B 0,C 180,E1 -15579.736,E2 -15579.736} C_VEL
LIN {X 0,Y 312.45,Z 387.639,A -85,B 0,C 180,E1 -15581.679,E2 -15581.679} C_VEL
LIN {X 0,Y 313.508,Z 380.756,A -85,B 0,C 180,E1 -15583.613,E2 -15583.613} C_VEL
LIN {X 0,Y 314.887,Z 372.14,A -85,B 0,C 180,E1 -15585.534,E2 -15585.534} C_VEL
